ELSE
	Cmd_R:=3;
END_CASE
END_ACTION
ACTION Command:
(* Default response OK/NODATA *)
Cmd_R:=0;
Cmd_RLen:=0;
TxLen:=16;

(* Check object *)
CASE Cmd_Obj OF

	EO_SYS:
		Cmd_SYS();
(*
	EO_GRU:
		Cmd_GRU();

	EO_PDC:
		Cmd_PDC();
*)
	EO_CAL:
		Cmd_CAL();

	EO_CRON:
		Cmd_CRON();

	EO_VRD:
		Cmd_VRD();

ELSE
	Cmd_R:=1;
END_CASE

(* Generate response *)
IF TxLen>0 THEN
	RAWTOHEX(ADR(Cmd_Obj)	,2,ADR(TxData[ 0]));
	RAWTOHEX(ADR(Cmd_ObjIdx),2,ADR(TxData[ 4]));
	RAWTOHEX(ADR(Cmd_R)		,2,ADR(TxData[ 8]));
	RAWTOHEX(ADR(Cmd_RLen)	,2,ADR(TxData[12]));
	TxTrig:=TRUE;
END_IF
END_ACTION

(* POU Utils Functions/TCPSERVER, ST *)
FUNCTION_BLOCK TCPSERVER
(***********************************************************************************************************	*)
(* Version: 1.6                                    			          											*)
(* Date: 11.02.2011                                   					          							    *)
(***********************************************************************************************************	*)
(* WAGO Kontakttechnik GmbH Hansastr. 27 32423 Minden(Westf.)													*)
(* Tel. +0049 571/887-0 Fax. +0049 571/887-0																	*)
(* Author: VB																									*)
(***********************************************************************************************************	*)
(*Description:	A TCP server to read and write data													       		*)
(*Historie:																										*)
(*Version 1.6: 11.02.2011: Changes according to 750-880/881											 			*)
(*Version 1.5: 27.11.2008 Bugfix allow reuse port																*)
(*Version 1.4: 13.10.2008 Bugfix transmitting large data														*)
(*Version 1.3: 15.01.2007 Changes according to FW11																*)
(*Version 1.2: 09.03.2006 Changes for socket handle 0											       			*)
(*Version 1.1: 14.02.2005 Release																				*)
(***********************************************************************************************************	*)
VAR CONSTANT
	STATE_INIT     				 : BYTE:= 0;
	STATE_OPEN     				 : BYTE:= 1;
	STATE_TX       				 : BYTE:= 20;
	STATE_RX       				 : BYTE:= 30;
	STATE_CLOSE    				 : BYTE:= 40;
	STATE_ERROR_TRAP		 	 : BYTE:= 200;
END_VAR
VAR_INPUT
	xEnable    					: BOOL;	 (* Set TRUE to enable function block *)
	wPortNumber					: WORD;  (* Port *)
	tServerTimeOut				: TIME:=t#50s;
	ptSendData					: POINTER TO ARRAY[0..MAX_SEND_TCP_SERVER] OF BYTE;
	diSendCount					: DINT;
END_VAR
VAR_OUTPUT
	xClientConnected  			: BOOL:= FALSE;
	diError 					: DINT:= 0;
END_VAR
(* Status Codes -----------------------------------------
	16#8001 => No socket descriptor available 
	16#8002 => SysSockBind fails 
	16#8003 => SysSockListen fails 
	16#8004 => switching to none blocking mode fails
	16#8005 => SysSockClose() returns FALSE 
    16#8006 => SysSockConnect() fails
    16#8007 => SysSockSend() fails
	16#8008 => error state machine 
	16#8009 => timeout while waiting for data from server 
	16#0001 => server waiting for client to establish connection
------------------------------------------------------------*)
VAR_IN_OUT
	xStartSend					: BOOL;
	aReceiveBuffer				: ARRAY [0..MAX_RECEIVE_TCP_SERVER] OF BYTE;
	diReceiveCount				: DINT;
END_VAR

VAR
	m_State    					: BYTE:= 0;
	m_ReceiveBuffer				: ARRAY [0..MAX_RECEIVE_TCP_SERVER_SOCKET] OF BYTE;
	m_ServerSocket				: DINT:= SOCKET_INVALID;
	m_Socket					: DINT:= SOCKET_INVALID;
	m_AddressInfo				: SOCKADDRESS;
	m_BytesReceived				: DINT;
	m_diReturn					: DINT;
	m_xReturn					: BOOL;
	m_SizeSockadr				: DWORD;
	m_ConnectionWatchdog		: TON;
	m_Flags						: DINT;
	m_NoneBlocking   			: DINT:= 1;
	m_Blocking   				: DINT:= 0;
	i							: INT;
	m_count						: DINT;
	diOption					: DINT := 1;
	on: DINT;
END_VAR
IF xEnable THEN
	CASE m_State OF
		STATE_INIT:
			(* Create Socket *)
			m_ServerSocket:= SysSockCreate( SOCKET_AF_INET, SOCKET_STREAM, 0);
			IF m_ServerSocket = SOCKET_INVALID THEN
				(* *)
				diError:= 16#8001;
				m_State:= STATE_ERROR_TRAP;
				RETURN;
			ELSE
				;
			END_IF
			(* Address bindings *)
			(********************)
			on:=1;
			SysSockSetOption( m_ServerSocket, SOCKET_SOL, SOCKET_SO_REUSEADDR, ADR(on), SIZEOF(on) );

			m_AddressInfo.sin_family:= SOCKET_AF_INET;
			m_AddressInfo.sin_port  := SysSockHtons( wPortNumber);
			m_AddressInfo.sin_addr  := SOCKET_INADDR_ANY;
			IF NOT SysSockBind( m_ServerSocket, ADR(m_AddressInfo), SIZEOF(m_AddressInfo)) THEN
				diError:= 16#8002;
				m_State:= STATE_ERROR_TRAP;
				RETURN;
			END_IF
			(* Wait for connections *)
			(************************)
			IF NOT SysSockListen( m_ServerSocket, 1) THEN
				diError:= 16#8003;
				m_State:= STATE_ERROR_TRAP;
			END_IF

			(* Puts SOCKET in NonBlocking mode *)
			m_diReturn:= SysSockIoctl( m_ServerSocket, SOCKET_FIONBIO, ADR(m_NoneBlocking));

			m_State:= STATE_OPEN;


		STATE_OPEN: 	(* Waiting for incomming connection *)
				m_SizeSockadr:=SIZEOF(m_AddressInfo);
				m_Socket:= SysSockAccept( m_ServerSocket, ADR(m_AddressInfo), ADR(m_SizeSockadr));
				diError:=State_open;
				IF m_Socket <> SOCKET_INVALID THEN
					xClientConnected:=TRUE;
					(*Set Push-Bit:new V1.5*)
					IF ADR(%MW0)=16#30000000  OR ADR(%MW0)=16#20000000 THEN (*841 or 881*)
						SysSockSetOption(
							diSocket:=m_Socket,
							diLevel:=6,
							diOption:=SOCKET_TCP_NODELAY,
							pOptionValue:=ADR(diOption),
							diOptionLength:=SIZEOF(diOption));
					ELSE
							;
					END_IF
					SysSockIoctl( m_Socket, SOCKET_FIONBIO, ADR(m_NoneBlocking));
					m_State:= STATE_RX;
					diError:=0;
				END_IF

		STATE_RX:
					m_BytesReceived:= SysSockRecv( m_Socket, ADR(m_ReceiveBuffer), SIZEOF(m_ReceiveBuffer), 0);
					CASE m_BytesReceived OF
					-1:(*no data available or error occured*)
						m_ConnectionWatchdog(IN:=TRUE , PT:=tServerTimeOut );
						IF m_connectionWatchdog.Q THEN
							m_State:= STATE_CLOSE;
							m_ConnectionWatchdog(IN:=FALSE);(*reset connection watchdog*)
							diError := 16#8009;
						END_IF
					0:(* socket was "gracefully closed"  *)
						m_State:= STATE_CLOSE;
						diError := 16#8003;
					ELSE
						(* Copy received data into receive buffer *)
						(********************************)
						FOR i:= 0 TO DINT_TO_INT(m_BytesReceived	)-1 DO
							aReceiveBuffer[diReceiveCount]:= m_ReceiveBuffer[i];
							diReceiveCount:=(diReceiveCount+1) MOD SIZEOF(aReceiveBuffer);
						END_FOR

						m_ConnectionWatchdog(IN:=FALSE);(*reset connection watchdog*)
					END_CASE

				(*send data*)
				IF xStartSend	 THEN
					m_State := STATE_TX;
				END_IF

	STATE_TX:	 (* send TCP-message *)
		m_diReturn := SysSockSend(diSocket := m_Socket,
								  pbyBuffer := ADR(ptSendData^[m_count]),(*geändert V1.4 bisher: [0] *)
								  diBufferSize := diSendCount-m_count,
								  diFlags :=m_Flags);
		CASE m_diReturn OF
		-1:	(* ERROR or data could not yet be send (V1.3 due to new FW11) *)
			m_ConnectionWatchdog(IN:=TRUE , PT:=tServerTimeOut );
			IF m_connectionWatchdog.Q THEN
				m_State:= STATE_CLOSE;
				m_ConnectionWatchdog(IN:=FALSE);(*reset connection watchdog*)
				diError := 16#8007;
			END_IF
		0: (* socket was "gracefully closed"  *)
			m_State := STATE_CLOSE;
			diError := 16#8003;
		ELSE (* succesful *)
			m_count:=m_count+m_diReturn;
			IF m_count>=diSendCount THEN
				diError := 16#0000;
				m_State := STATE_RX;
				m_count:=0;
				xStartSend:=FALSE;
			END_IF
			m_ConnectionWatchdog(IN:=FALSE);(*reset connection watchdog*)
		END_CASE


		STATE_CLOSE:	(* Close the server *)

		IF ADR(%MW0)=16#30000000  OR ADR(%MW0)=16#20000000 THEN (*841 or 881*)
			;
		ELSE
			IF m_Socket>=0 THEN
				SysSockShutdown(m_Socket, 0);;(*870*)
			END_IF
		END_IF
		IF m_Socket>=0 THEN
			SysSockClose( m_Socket);
		END_IF
		xClientConnected:= FALSE;
		m_State:= STATE_OPEN; (* Try to open the server again *)
		m_ConnectionWatchdog(IN:=FALSE);(*reset connection watchdog*)

		STATE_ERROR_TRAP: (* Error Read/Write socket  *)
			m_State:= STATE_ERROR_TRAP;

	ELSE  (* Bad FSM code trap  *)
			m_State:= STATE_ERROR_TRAP;
			diError:= 16#8008;
	END_CASE;
ELSE
	IF m_State <> STATE_INIT THEN
		IF ADR(%MW0)=16#30000000  OR ADR(%MW0)=16#20000000 THEN (*841 or 881*)
			;
		ELSE
			IF m_Socket>=0 THEN
				SysSockShutdown(m_Socket, 0);;(*870*)
			END_IF
		END_IF
		IF m_Socket>=0 THEN
			SysSockClose( m_Socket);
		END_IF
		IF ADR(%MW0)=16#30000000  OR ADR(%MW0)=16#20000000 THEN (*841 or 881*)
			;
		ELSE
			IF m_ServerSocket>=0 THEN
				SysSockShutdown(m_ServerSocket, 0);;(*870*)
			END_IF
		END_IF
		IF m_ServerSocket>=0 THEN
			SysSockClose( m_ServerSocket);
		END_IF
		xClientConnected:= FALSE;
		diError:= 0;
		m_State:= STATE_init; (* Try to open the server again *)
		m_ConnectionWatchdog(IN:=FALSE);(*reset connection watchdog*)
	END_IF
END_IF
END_FUNCTION_BLOCK

(* POU Utils Functions/HEXTORAW, ST *)
FUNCTION HEXTORAW : WORD
VAR_INPUT
	pString		: POINTER TO BYTE;
	StringLen	: WORD;
	pData		: POINTER TO BYTE;
END_VAR
VAR
	xl: WORD;
	xi: WORD;
	xr: BYTE;
END_VAR
xl:=0;
xi:=0;

WHILE xi<StringLen DO

	IF pString^>=97 AND pString^<=102 THEN
		xr := pString^ - 87;
	ELSIF pString^>=65 AND pString^<=70 THEN
		xr := pString^ - 55;
	ELSIF pString^>=48 AND pString^<=57 THEN
		xr := pString^ - 48;
	ELSE
		xr := 16;
	END_IF

	IF xr<16 THEN
		IF (xi AND 1)=0 THEN
			pData^ := xr * 16;
		ELSE
			pData^ := pData^ + xr;
			pData := pData + 1;
			xl := xl + 1;
		END_IF
	END_IF

	xi := xi + 1;
	pString := pString + 1;

END_WHILE

HEXTORAW:=xl;
END_FUNCTION

(* POU Utils Functions/RAWTOHEX, ST *)
FUNCTION RAWTOHEX : WORD
VAR_INPUT
	pData: POINTER TO BYTE;
	DataLen: WORD;
	pString: POINTER TO BYTE;
END_VAR
VAR
	xl: WORD;
END_VAR
xl:=0;

WHILE DataLen>0 DO

	pString^ := (pData^ / 16#10) + 48 + (((pData^ / 16#10)/10)*7);
	pString:=pString+1;
	pString^ := (pData^ AND 16#0F)  + 48 + (((pData^ AND 16#0F)/10)*7);
	pString:=pString+1;
	pData:=pData+1;
	DataLen:=DataLen-1;
	xl:=xl+2;

END_WHILE

(*pString^:=0;*)

RAWTOHEX:=xl;
END_FUNCTION

(* POU Utils/USRLED_Update, ST *)
PROGRAM USRLED_Update
VAR
	OldStatus: en_SYS_Status;

	aFS : ARRAY [0..24] OF FLASHING_SEQUENCE :=
		(Colour:=GREEN,  Frequency:=1,   Relation:=128, Duration:=t#0s,    NextIndex:=0),  (* 0 => RUNNING *)
		(Colour:=ORANGE, Frequency:=1,   Relation:=128, Duration:=t#0s,    NextIndex:=1),  (* 1 => INIT *)
		(Colour:=RED,    Frequency:=4,   Relation:=128, Duration:=t#0s,    NextIndex:=2),  (* 2 => ERROR *)
		(Colour:=RED,    Frequency:=10,  Relation:=128, Duration:=t#0s,    NextIndex:=3),  (* 3 => ALARM *)
		(Colour:=ORANGE, Frequency:=200, Relation:=16,  Duration:=t#100ms, NextIndex:=11), (* 10 *)
		(Colour:=ORANGE, Frequency:=200, Relation:=32,  Duration:=t#100ms, NextIndex:=12),
		(Colour:=ORANGE, Frequency:=200, Relation:=64,  Duration:=t#100ms, NextIndex:=13),
		(Colour:=ORANGE, Frequency:=200, Relation:=128, Duration:=t#100ms, NextIndex:=14),
		(Colour:=ORANGE, Frequency:=200, Relation:=192, Duration:=t#100ms, NextIndex:=15),
		(Colour:=ORANGE, Frequency:=200, Relation:=128, Duration:=t#100ms, NextIndex:=16),
		(Colour:=ORANGE, Frequency:=200, Relation:=64,  Duration:=t#100ms, NextIndex:=17),
		(Colour:=ORANGE, Frequency:=200, Relation:=32,  Duration:=t#100ms, NextIndex:=18),
		(Colour:=ORANGE, Frequency:=200, Relation:=16,  Duration:=t#100ms, NextIndex:=19),
		(Colour:=ORANGE, Frequency:=200, Relation:=8,   Duration:=t#100ms, NextIndex:=10),
		(Colour:=GREEN,  Frequency:=200, Relation:=16,  Duration:=t#100ms, NextIndex:=21), (* 20 *)
		(Colour:=GREEN,  Frequency:=200, Relation:=32,  Duration:=t#100ms, NextIndex:=22),
		(Colour:=GREEN,  Frequency:=200, Relation:=64,  Duration:=t#100ms, NextIndex:=23),
		(Colour:=GREEN,  Frequency:=200, Relation:=128, Duration:=t#100ms, NextIndex:=24),
		(Colour:=GREEN,  Frequency:=200, Relation:=192, Duration:=t#100ms, NextIndex:=25),
		(Colour:=GREEN,  Frequency:=200, Relation:=128, Duration:=t#100ms, NextIndex:=26),
		(Colour:=GREEN,  Frequency:=200, Relation:=64,  Duration:=t#100ms, NextIndex:=27),
		(Colour:=GREEN,  Frequency:=200, Relation:=32,  Duration:=t#100ms, NextIndex:=28),
		(Colour:=GREEN,  Frequency:=200, Relation:=16,  Duration:=t#100ms, NextIndex:=29),
		(Colour:=GREEN,  Frequency:=200, Relation:=8,   Duration:=t#100ms, NextIndex:=20);

	pFS : POINTER TO FLASHING_SEQUENCE;


END_VAR
IF Sys.Status <> OldStatus THEN

	OldStatus:=Sys.Status;

	CASE OldStatus OF

		S_STARTUP:
			pFS:=ADR(aFS);
			SET_FLASHING_SEQUENCE(EN:=TRUE, POINTER_TO_POINTER_TO_ARRAY:=ADR(pFS));
			SET_FLASHING_SEQUENCE_INDEX(EN:=TRUE, IMMEDIATE:=FALSE, INDEX:=1);
			START_FLASHING_SEQUENCE(EN:=TRUE);

		S_RUNNING:
			SET_FLASHING_SEQUENCE_INDEX(EN:=TRUE, IMMEDIATE:=TRUE, INDEX:=0);

	END_CASE

END_IF
END_PROGRAM

(* POU Utils/CSV_Log, ST *)
FUNCTION CSV_Log : BOOL
VAR_INPUT
END_VAR
VAR CONSTANT
	LogFileName:STRING:='S:\LOGS_ID4V3.CSV';
END_VAR
VAR
	s1 : STRING(256);
	hFile: 	DWORD;
END_VAR
(* Check file presence *)
hFile:=SysFileOpen(LogFileName,'r');
IF hFile=0 THEN
	(*** File not exist *** Create file and write header *)
	hFile:=SysFileOpen(LogFileName,'w');
	IF hFile<>0 THEN
		(* Write CSV header *)
		s1:='Title1;Title2,...';
		SysFileWrite(hFile, ADR(s1), LEN(s1));
		SysFileWrite(hFile, ADR(Logger_CRLF), LEN(Logger_CRLF));
	END_IF
ELSE
	(*** File exist *** Close file and reopen in append mode *)
	SysFileClose(hFile);
	hFile:=SysFileOpen(LogFileName,'a');
END_IF

(* Log to file *)
IF hFile<>0 THEN
	(* Date stamp *)
	s1:=REPLACE( Sys.Time_LogString , ' ' , 1 , 11 );
	SysFileWrite(hFile, ADR(s1), LEN(s1));
	(* Write CSV data *)
	s1:=CONCAT(';', 'Data1' );
	s1:=CONCAT(s1 , ';');
	s1:=CONCAT(s1 , 'Data2' );
	s1:=CONCAT(s1 , ';');
	s1:=CONCAT(s1 , '...' );
	SysFileWrite(hFile, ADR(s1), LEN(s1));
	(* Add line CRLF and close *)
	SysFileWrite(hFile, ADR(Logger_CRLF), LEN(Logger_CRLF));
	SysFileClose(hFile);
END_IF
END_FUNCTION

(* POU CLV/CLV__Cmd, ST *)
PROGRAM CLV__Cmd
(* === Execute server command ===
   v1.0[27/05/15]
*)
VAR_INPUT
END_VAR
VAR_OUTPUT
	Cmd_R
	Cmd_RLen
END_VAR
VAR
END_VAR
(* Default response OK/NODATA *)
Cmd_R:=0;
Cmd_RLen:=0;
TxLen:=16;

(* Check object *)
CASE Cmd_Obj OF

	EO_SYS:
		Cmd_SYS();
(*
	EO_GRU:
		Cmd_GRU();

	EO_PDC:
		Cmd_PDC();

	EO_CAL:
		Cmd_CAL();

	EO_CRON:
		Cmd_CRON();
*)
ELSE
	Cmd_R:=1;
END_CASE
END_PROGRAM

(* POU CLV/CLV__LogTrig, ST *)
PROGRAM CLV__LogTrig
(* === Log regular informations ===
   v1.0[27/05/15]
*)
VAR
	s1 : STRING(160);
	i  : BYTE;
END_VAR
(*---------------------------------------------------------------*)
	CLV.LogHead();
(*---------------------------------------------------------------*)

(*** PROJECT SPECIFIC CODE HERE ***)

(*---------------------------------------------------------------*)
	CLV.LogSend();
(*---------------------------------------------------------------*)
END_PROGRAM

(* POU Plant/SCA_Proc, ST *)
PROGRAM SCA_Proc
VAR
	SCA01_5			:FLT_TAP;
	SCA01_6			:FLT_TAP;

	SCA02_1			:FLT_TAP;
	SCA02_2			:FLT_TAP;
	SCA02_3			:FLT_TAP;
	SCA02_4			:FLT_TAP;
	SCA02_5			:FLT_TAP;
	SCA02_6			:FLT_TAP;
	SCA02_7			:FLT_TAP;
	SCA02_8			:FLT_TAP;
	SCA02_9			:FLT_TAP;

	SCA03_1			:FLT_TAP;
	SCA03_2			:FLT_TAP;
	SCA03_3			:FLT_TAP;
	SCA03_4			:FLT_TAP;
	SCA03_5			:FLT_TAP;
	SCA03_6			:FLT_TAP;
	SCA03_7			:FLT_TAP;
	SCA03_8			:FLT_TAP;
	SCA03_9			:FLT_TAP;
	SCA03_10		:FLT_TAP;
	SCA03_11		:FLT_TAP;
	SCA03_12		:FLT_TAP;
	SCA03_13		:FLT_TAP;
	SCA03_14		:FLT_TAP;
	SCA03_15		:FLT_TAP;
	SCA03_16		:FLT_TAP;
	SCA03_17		:FLT_TAP;
	SCA03_18		:FLT_TAP;
	SCA03_19		:FLT_TAP;
	SCA03_20		:FLT_TAP;
	SCA03_21		:FLT_TAP;
	SCA03_22		:FLT_TAP;

END_VAR
(***** SCA01 *****)
SCA01_1_DO:=SCA01_6.OUT;

SCA01_2_DO:=SCA02_1.OUT;

SCA01_3_DO:=SCA02_2.OUT  OR SCA02_3.OUT  OR SCA02_4.OUT  OR SCA02_5.OUT  OR SCA02_6.OUT  OR
			SCA02_7.OUT  OR SCA02_8.OUT  OR SCA02_9.OUT;

SCA01_4_DO:=SCA03_1.OUT  OR SCA03_2.OUT  OR SCA03_3.OUT  OR SCA03_4.OUT  OR SCA03_5.OUT  OR
			SCA03_6.OUT  OR SCA03_7.OUT  OR SCA03_8.OUT  OR SCA03_9.OUT  OR SCA03_10.OUT OR
			SCA03_11.OUT OR SCA03_12.OUT OR SCA03_13.OUT OR SCA03_14.OUT OR SCA03_15.OUT OR
			SCA03_16.OUT OR SCA03_17.OUT OR SCA03_18.OUT OR SCA03_19.OUT OR SCA03_20.OUT OR
			SCA03_21.OUT OR SCA03_22.OUT;

SCA01_5(IN:=SCA01_5_DI);
IF SCA01_5.EVL THEN LogEv(EL_Wrn,EO_SCA,1,1,'5'); END_IF
IF SCA01_5.EVH THEN	LogEv(EL_Log,EO_SCA,1,2,'5'); END_IF

SCA01_6(IN:=SCA01_6_DI);
IF SCA01_6.EVL THEN	LogEv(EL_Wrn,EO_SCA,1,1,'6'); END_IF
IF SCA01_6.EVH THEN	LogEv(EL_Log,EO_SCA,1,2,'6'); END_IF

(***** SCA02 *****)

SCA02_1(IN:=SCA02_1_DI);
IF SCA02_1.EVL THEN	LogEv(EL_Wrn,EO_SCA,2,1,'1'); END_IF
IF SCA02_1.EVH THEN	LogEv(EL_Log,EO_SCA,2,2,'1'); END_IF
SCA02_2(IN:=SCA02_2_DI);
IF SCA02_2.EVL THEN	LogEv(EL_Wrn,EO_SCA,2,1,'2'); END_IF
IF SCA02_2.EVH THEN	LogEv(EL_Log,EO_SCA,2,2,'2'); END_IF
SCA02_3(IN:=SCA02_3_DI);
IF SCA02_3.EVL THEN	LogEv(EL_Wrn,EO_SCA,2,1,'3'); END_IF
IF SCA02_3.EVH THEN	LogEv(EL_Log,EO_SCA,2,2,'3'); END_IF
SCA02_4(IN:=SCA02_4_DI);
IF SCA02_4.EVL THEN	LogEv(EL_Wrn,EO_SCA,2,1,'4'); END_IF
IF SCA02_4.EVH THEN	LogEv(EL_Log,EO_SCA,2,2,'4'); END_IF
SCA02_5(IN:=SCA02_5_DI);
IF SCA02_5.EVL THEN	LogEv(EL_Wrn,EO_SCA,2,1,'5'); END_IF
IF SCA02_5.EVH THEN	LogEv(EL_Log,EO_SCA,2,2,'5'); END_IF
SCA02_6(IN:=SCA02_6_DI);
IF SCA02_6.EVL THEN	LogEv(EL_Wrn,EO_SCA,2,1,'6'); END_IF
IF SCA02_6.EVH THEN	LogEv(EL_Log,EO_SCA,2,2,'6'); END_IF
SCA02_7(IN:=SCA02_7_DI);
IF SCA02_7.EVL THEN	LogEv(EL_Wrn,EO_SCA,2,1,'7'); END_IF
IF SCA02_7.EVH THEN	LogEv(EL_Log,EO_SCA,2,2,'7'); END_IF
SCA02_8(IN:=SCA02_8_DI);
IF SCA02_8.EVL THEN	LogEv(EL_Wrn,EO_SCA,2,1,'8'); END_IF
IF SCA02_8.EVH THEN	LogEv(EL_Log,EO_SCA,2,2,'8'); END_IF
SCA02_9(IN:=SCA02_9_DI);
IF SCA02_9.EVL THEN	LogEv(EL_Wrn,EO_SCA,2,1,'9'); END_IF
IF SCA02_9.EVH THEN	LogEv(EL_Log,EO_SCA,2,2,'9'); END_IF

(***** SCA03 *****)

SCA03_1(IN:=SCA03_1_DI);
IF SCA03_1.EVL THEN	LogEv(EL_Wrn,EO_SCA,3,1,'1'); END_IF
IF SCA03_1.EVH THEN	LogEv(EL_Log,EO_SCA,3,2,'1'); END_IF
SCA03_2(IN:=SCA03_2_DI);
IF SCA03_2.EVL THEN	LogEv(EL_Wrn,EO_SCA,3,1,'2'); END_IF
IF SCA03_2.EVH THEN	LogEv(EL_Log,EO_SCA,3,2,'2'); END_IF
SCA03_3(IN:=SCA03_3_DI);
IF SCA03_3.EVL THEN	LogEv(EL_Wrn,EO_SCA,3,1,'3'); END_IF
IF SCA03_3.EVH THEN	LogEv(EL_Log,EO_SCA,3,2,'3'); END_IF
SCA03_4(IN:=SCA03_4_DI);
IF SCA03_4.EVL THEN	LogEv(EL_Wrn,EO_SCA,3,1,'4'); END_IF
IF SCA03_4.EVH THEN	LogEv(EL_Log,EO_SCA,3,2,'4'); END_IF
SCA03_5(IN:=SCA03_5_DI);
IF SCA03_5.EVL THEN	LogEv(EL_Wrn,EO_SCA,3,1,'5'); END_IF
IF SCA03_5.EVH THEN	LogEv(EL_Log,EO_SCA,3,2,'5'); END_IF
SCA03_6(IN:=SCA03_6_DI);
IF SCA03_6.EVL THEN	LogEv(EL_Wrn,EO_SCA,3,1,'6'); END_IF
IF SCA03_6.EVH THEN	LogEv(EL_Log,EO_SCA,3,2,'6'); END_IF
SCA03_7(IN:=SCA03_7_DI);
IF SCA03_7.EVL THEN	LogEv(EL_Wrn,EO_SCA,3,1,'7'); END_IF
IF SCA03_7.EVH THEN	LogEv(EL_Log,EO_SCA,3,2,'7'); END_IF
SCA03_8(IN:=SCA03_8_DI);
IF SCA03_8.EVL THEN	LogEv(EL_Wrn,EO_SCA,3,1,'8'); END_IF
IF SCA03_8.EVH THEN	LogEv(EL_Log,EO_SCA,3,2,'8'); END_IF
SCA03_9(IN:=SCA03_9_DI);
IF SCA03_9.EVL THEN	LogEv(EL_Wrn,EO_SCA,3,1,'9'); END_IF
IF SCA03_9.EVH THEN	LogEv(EL_Log,EO_SCA,3,2,'9'); END_IF
SCA03_10(IN:=SCA03_10_DI);
IF SCA03_10.EVL THEN	LogEv(EL_Wrn,EO_SCA,3,1,'10'); END_IF
IF SCA03_10.EVH THEN	LogEv(EL_Log,EO_SCA,3,2,'10'); END_IF
SCA03_11(IN:=SCA03_11_DI);
IF SCA03_11.EVL THEN	LogEv(EL_Wrn,EO_SCA,3,1,'11'); END_IF
IF SCA03_11.EVH THEN	LogEv(EL_Log,EO_SCA,3,2,'11'); END_IF
SCA03_12(IN:=SCA03_12_DI);
IF SCA03_12.EVL THEN	LogEv(EL_Wrn,EO_SCA,3,1,'12'); END_IF
IF SCA03_12.EVH THEN	LogEv(EL_Log,EO_SCA,3,2,'12'); END_IF
SCA03_13(IN:=SCA03_13_DI);
IF SCA03_13.EVL THEN	LogEv(EL_Wrn,EO_SCA,3,1,'13'); END_IF
IF SCA03_13.EVH THEN	LogEv(EL_Log,EO_SCA,3,2,'13'); END_IF
SCA03_14(IN:=SCA03_14_DI);
IF SCA03_14.EVL THEN	LogEv(EL_Wrn,EO_SCA,3,1,'14'); END_IF
IF SCA03_14.EVH THEN	LogEv(EL_Log,EO_SCA,3,2,'14'); END_IF
SCA03_15(IN:=SCA03_15_DI);
IF SCA03_15.EVL THEN	LogEv(EL_Wrn,EO_SCA,3,1,'15'); END_IF
IF SCA03_15.EVH THEN	LogEv(EL_Log,EO_SCA,3,2,'15'); END_IF
SCA03_16(IN:=SCA03_16_DI);
IF SCA03_16.EVL THEN	LogEv(EL_Wrn,EO_SCA,3,1,'16'); END_IF
IF SCA03_16.EVH THEN	LogEv(EL_Log,EO_SCA,3,2,'16'); END_IF
SCA03_17(IN:=SCA03_17_DI);
IF SCA03_17.EVL THEN	LogEv(EL_Wrn,EO_SCA,3,1,'17'); END_IF
IF SCA03_17.EVH THEN	LogEv(EL_Log,EO_SCA,3,2,'17'); END_IF
SCA03_18(IN:=SCA03_18_DI);
IF SCA03_18.EVL THEN	LogEv(EL_Wrn,EO_SCA,3,1,'18'); END_IF
IF SCA03_18.EVH THEN	LogEv(EL_Log,EO_SCA,3,2,'18'); END_IF
SCA03_19(IN:=SCA03_19_DI);
IF SCA03_19.EVL THEN	LogEv(EL_Wrn,EO_SCA,3,1,'19'); END_IF
IF SCA03_19.EVH THEN	LogEv(EL_Log,EO_SCA,3,2,'19'); END_IF
SCA03_20(IN:=SCA03_20_DI);
IF SCA03_20.EVL THEN	LogEv(EL_Wrn,EO_SCA,3,1,'20'); END_IF
IF SCA03_20.EVH THEN	LogEv(EL_Log,EO_SCA,3,2,'20'); END_IF
SCA03_21(IN:=SCA03_21_DI);
IF SCA03_21.EVL THEN	LogEv(EL_Wrn,EO_SCA,3,1,'21'); END_IF
IF SCA03_21.EVH THEN	LogEv(EL_Log,EO_SCA,3,2,'21'); END_IF
SCA03_22(IN:=SCA03_22_DI);
IF SCA03_22.EVL THEN	LogEv(EL_Wrn,EO_SCA,3,1,'22'); END_IF
IF SCA03_22.EVH THEN	LogEv(EL_Log,EO_SCA,3,2,'22'); END_IF
END_PROGRAM
ACTION AddLogData:
Logger.s1:='&SCA01=';
Logger.s1:=CONCAT(Logger.s1,BYTE_TO_STRING(BOOL_TO_BYTE(SCA01_1_DO))		); Logger.s1:=CONCAT(Logger.s1,';');
Logger.s1:=CONCAT(Logger.s1,BYTE_TO_STRING(BOOL_TO_BYTE(SCA01_2_DO))		); Logger.s1:=CONCAT(Logger.s1,';');
Logger.s1:=CONCAT(Logger.s1,BYTE_TO_STRING(BOOL_TO_BYTE(SCA01_3_DO))		); Logger.s1:=CONCAT(Logger.s1,';');
Logger.s1:=CONCAT(Logger.s1,BYTE_TO_STRING(BOOL_TO_BYTE(SCA01_4_DO))		); Logger.s1:=CONCAT(Logger.s1,';');
Logger.s1:=CONCAT(Logger.s1,BYTE_TO_STRING(BOOL_TO_BYTE(SCA01_5.OUT))		); Logger.s1:=CONCAT(Logger.s1,';');
Logger.s1:=CONCAT(Logger.s1,BYTE_TO_STRING(BOOL_TO_BYTE(SCA01_6.OUT))		);
ADDSTRING(ADR(Logger.TData), ADR(Logger.s1), Logger.TLen);

Logger.s1:='&SCA02=';
Logger.s1:=CONCAT(Logger.s1,BYTE_TO_STRING(BOOL_TO_BYTE(SCA02_1.OUT))		); Logger.s1:=CONCAT(Logger.s1,';');
Logger.s1:=CONCAT(Logger.s1,BYTE_TO_STRING(BOOL_TO_BYTE(SCA02_2.OUT))		); Logger.s1:=CONCAT(Logger.s1,';');
Logger.s1:=CONCAT(Logger.s1,BYTE_TO_STRING(BOOL_TO_BYTE(SCA02_3.OUT))		); Logger.s1:=CONCAT(Logger.s1,';');
Logger.s1:=CONCAT(Logger.s1,BYTE_TO_STRING(BOOL_TO_BYTE(SCA02_4.OUT))		); Logger.s1:=CONCAT(Logger.s1,';');
Logger.s1:=CONCAT(Logger.s1,BYTE_TO_STRING(BOOL_TO_BYTE(SCA02_5.OUT))		); Logger.s1:=CONCAT(Logger.s1,';');
Logger.s1:=CONCAT(Logger.s1,BYTE_TO_STRING(BOOL_TO_BYTE(SCA02_6.OUT))		); Logger.s1:=CONCAT(Logger.s1,';');
Logger.s1:=CONCAT(Logger.s1,BYTE_TO_STRING(BOOL_TO_BYTE(SCA02_7.OUT))		); Logger.s1:=CONCAT(Logger.s1,';');
Logger.s1:=CONCAT(Logger.s1,BYTE_TO_STRING(BOOL_TO_BYTE(SCA02_8.OUT))		); Logger.s1:=CONCAT(Logger.s1,';');
Logger.s1:=CONCAT(Logger.s1,BYTE_TO_STRING(BOOL_TO_BYTE(SCA02_9.OUT))		);
ADDSTRING(ADR(Logger.TData), ADR(Logger.s1), Logger.TLen);

Logger.s1:='&SCA03=';
Logger.s1:=CONCAT(Logger.s1,BYTE_TO_STRING(BOOL_TO_BYTE(SCA03_1.OUT))		); Logger.s1:=CONCAT(Logger.s1,';');
Logger.s1:=CONCAT(Logger.s1,BYTE_TO_STRING(BOOL_TO_BYTE(SCA03_2.OUT))		); Logger.s1:=CONCAT(Logger.s1,';');
Logger.s1:=CONCAT(Logger.s1,BYTE_TO_STRING(BOOL_TO_BYTE(SCA03_3.OUT))		); Logger.s1:=CONCAT(Logger.s1,';');
Logger.s1:=CONCAT(Logger.s1,BYTE_TO_STRING(BOOL_TO_BYTE(SCA03_4.OUT))		); Logger.s1:=CONCAT(Logger.s1,';');
Logger.s1:=CONCAT(Logger.s1,BYTE_TO_STRING(BOOL_TO_BYTE(SCA03_5.OUT))		); Logger.s1:=CONCAT(Logger.s1,';');
Logger.s1:=CONCAT(Logger.s1,BYTE_TO_STRING(BOOL_TO_BYTE(SCA03_6.OUT))		); Logger.s1:=CONCAT(Logger.s1,';');
Logger.s1:=CONCAT(Logger.s1,BYTE_TO_STRING(BOOL_TO_BYTE(SCA03_7.OUT))		); Logger.s1:=CONCAT(Logger.s1,';');
Logger.s1:=CONCAT(Logger.s1,BYTE_TO_STRING(BOOL_TO_BYTE(SCA03_8.OUT))		); Logger.s1:=CONCAT(Logger.s1,';');
Logger.s1:=CONCAT(Logger.s1,BYTE_TO_STRING(BOOL_TO_BYTE(SCA03_9.OUT))		); Logger.s1:=CONCAT(Logger.s1,';');
Logger.s1:=CONCAT(Logger.s1,BYTE_TO_STRING(BOOL_TO_BYTE(SCA03_10.OUT))		); Logger.s1:=CONCAT(Logger.s1,';');
Logger.s1:=CONCAT(Logger.s1,BYTE_TO_STRING(BOOL_TO_BYTE(SCA03_11.OUT))		); Logger.s1:=CONCAT(Logger.s1,';');
Logger.s1:=CONCAT(Logger.s1,BYTE_TO_STRING(BOOL_TO_BYTE(SCA03_12.OUT))		); Logger.s1:=CONCAT(Logger.s1,';');
Logger.s1:=CONCAT(Logger.s1,BYTE_TO_STRING(BOOL_TO_BYTE(SCA03_13.OUT))		); Logger.s1:=CONCAT(Logger.s1,';');
Logger.s1:=CONCAT(Logger.s1,BYTE_TO_STRING(BOOL_TO_BYTE(SCA03_14.OUT))		); Logger.s1:=CONCAT(Logger.s1,';');
Logger.s1:=CONCAT(Logger.s1,BYTE_TO_STRING(BOOL_TO_BYTE(SCA03_15.OUT))		); Logger.s1:=CONCAT(Logger.s1,';');
Logger.s1:=CONCAT(Logger.s1,BYTE_TO_STRING(BOOL_TO_BYTE(SCA03_16.OUT))		); Logger.s1:=CONCAT(Logger.s1,';');
Logger.s1:=CONCAT(Logger.s1,BYTE_TO_STRING(BOOL_TO_BYTE(SCA03_17.OUT))		); Logger.s1:=CONCAT(Logger.s1,';');
Logger.s1:=CONCAT(Logger.s1,BYTE_TO_STRING(BOOL_TO_BYTE(SCA03_18.OUT))		); Logger.s1:=CONCAT(Logger.s1,';');
Logger.s1:=CONCAT(Logger.s1,BYTE_TO_STRING(BOOL_TO_BYTE(SCA03_19.OUT))		); Logger.s1:=CONCAT(Logger.s1,';');
Logger.s1:=CONCAT(Logger.s1,BYTE_TO_STRING(BOOL_TO_BYTE(SCA03_20.OUT))		); Logger.s1:=CONCAT(Logger.s1,';');
Logger.s1:=CONCAT(Logger.s1,BYTE_TO_STRING(BOOL_TO_BYTE(SCA03_21.OUT))		); Logger.s1:=CONCAT(Logger.s1,';');
Logger.s1:=CONCAT(Logger.s1,BYTE_TO_STRING(BOOL_TO_BYTE(SCA03_22.OUT))		);
ADDSTRING(ADR(Logger.TData), ADR(Logger.s1), Logger.TLen);
END_ACTION

(* POU Utils Functions/FLT_TAP, ST *)
FUNCTION_BLOCK FLT_TAP
VAR_INPUT
	IN		: BOOL;
	TAP		: BYTE:=4;
	INITEV	: BOOL:=TRUE;
END_VAR
VAR_OUTPUT
	OUT		: BOOL;
	EVH		: BOOL;
	EVL		: BOOL;
END_VAR
VAR
	init	: BOOL:=FALSE;
	cnt		: BYTE;
END_VAR
EVH:=FALSE;
EVL:=FALSE;

IF NOT init THEN
	init := TRUE;
	IF INITEV THEN
		OUT  := NOT IN;
		cnt  := TAP;
	ELSE
		OUT  := IN;
	END_IF
END_IF

IF OUT<>IN THEN
	cnt:=cnt+1;
	IF cnt>TAP THEN
		OUT:=IN;
		cnt:=0;
		IF OUT THEN EVH:=TRUE; ELSE EVL:=TRUE; END_IF
	END_IF
ELSE
	cnt:=0;
END_IF
END_FUNCTION_BLOCK

(* POU TCP_Logger/LogEv, ST *)
FUNCTION LogEv : BOOL
VAR_INPUT
	Level	: en_Logger_ErrLev;
	Object  : en_SYS_Objects;
	Index	: WORD;
	Error	: WORD;
	Message : STRING;
END_VAR
VAR
	s1 : STRING(160);
	i  : INT;
END_VAR
(* Execute error level operations *)
CASE Level OF
	EL_Wrn: 		Sys.Warning:=TRUE;
	EL_Alarm: 		Sys.Alarm  :=TRUE;
	EL_AlarmStop: 	Sys.Alarm  :=TRUE; (* GO TO STOP STATE!! *)
END_CASE

(* Fill lastlog list *)
s1:=CONCAT(Sys.Time_LogString,';Lev=');
s1:=CONCAT(s1,INT_TO_STRING(Level));
s1:=CONCAT(s1,';Obj=');
s1:=CONCAT(s1,INT_TO_STRING(Object));
s1:=CONCAT(s1,';Idx=');
s1:=CONCAT(s1,WORD_TO_STRING(Index));
s1:=CONCAT(s1,';Err=');
s1:=CONCAT(s1,WORD_TO_STRING(Error));
Sys.LastLogs_Dat[Sys.LastLogs_Idx]:=s1;
Sys.LastLogs_Msg[Sys.LastLogs_Idx]:=Message;
Sys.LastLogs_Idx:=Sys.LastLogs_Idx+1;
IF Sys.LastLogs_Idx>5 THEN Sys.LastLogs_Idx:=0; END_IF

(*---------------------------------------------------------------*)
	Logger_Head();
(*---------------------------------------------------------------*)

(* Insert ERR *)
s1:=CONCAT('&ERR=',INT_TO_STRING(Level));
s1:=CONCAT(s1,';');
s1:=CONCAT(s1,INT_TO_STRING(Object));
s1:=CONCAT(s1,';');
s1:=CONCAT(s1,WORD_TO_STRING(Index));
s1:=CONCAT(s1,';');
s1:=CONCAT(s1,WORD_TO_STRING(Error));
s1:=CONCAT(s1,';');
ADDSTRING(ADR(Logger.TData), ADR(s1), Logger.TLen);
s1:=Message;
STR_NOSPACES(ADR(s1));
ADDSTRING(ADR(Logger.TData), ADR(s1), Logger.TLen);

(*---------------------------------------------------------------*)
	Logger_Send();
(*---------------------------------------------------------------*)
END_FUNCTION

(* POU TCP_Logger/Logger_Head, ST *)
FUNCTION Logger_Head : BOOL
VAR
	s1 : STRING(160);
	i  : BYTE;
END_VAR
Logger.TLen:=0;
(* Set GET header *)
ADDSTRING(ADR(Logger.TData), ADR(Logger_GETSTART), Logger.TLen);

(* Insert Header *)
s1:=INSERT('ID=&V=1&D=',DWORD_TO_STRING(Plant_SN),3);
s1:=CONCAT(s1,Sys.Time_LogString);
s1:=CONCAT(s1,'&S=');
IF Sys.Alarm THEN i:=2; ELSIF Sys.Warning THEN i:=1; ELSE i:=0; END_IF
s1:=CONCAT(s1,BYTE_TO_STRING(i));
ADDSTRING(ADR(Logger.TData), ADR(s1), Logger.TLen);
END_FUNCTION

(* POU Utils Functions/ADDSTRING, ST *)
FUNCTION ADDSTRING : BOOL (* Append string to a byte buffer *)
VAR_INPUT
	pTxData: POINTER TO BYTE;
	pString: POINTER TO BYTE;
END_VAR
VAR_IN_OUT
	TxLen: DINT;
END_VAR
VAR
END_VAR
pTxData:=pTxData+TxLen;
WHILE pString^<>0 DO
	pTxData^:=pString^;
	pString:=pString+1;
	pTxData:=pTxData+1;
	TxLen:=TxLen+1;
END_WHILE
END_FUNCTION

(* POU Utils Functions/STR_NOSPACES, ST *)
FUNCTION STR_NOSPACES : BOOL (* Replace spaces and bad chars with allowed ones, used as HTTP-GET validator *)
VAR_INPUT
	pString: POINTER TO BYTE;
END_VAR
VAR
END_VAR
WHILE pString^<>0 DO
	IF pString^=16#20 (* space *) THEN pString^:=16#5F; (*'_'*) END_IF
	pString:=pString+1;
END_WHILE
END_FUNCTION

(* POU TCP_Logger/Logger_Send, ST *)
FUNCTION Logger_Send : BOOL
VAR
	hFile: 	DWORD;
	pos:	DWORD;
END_VAR
(* Finalize string *)
ADDSTRING(ADR(Logger.TData), ADR(Logger_GETEND), Logger.TLen);

(* Read log position *)
pos:=SysFileGetSize(Logger_DataFile);
(* Check log size, bckup and erase if no pending messages *)
IF pos>5000000(*5M*) THEN
	hFile:=SysFileOpen(Logger_IndexFile,'r');
	IF hFile=0 THEN
		SysFileDelete(Logger_DataFileOld);
		SysFileRename(Logger_DataFile,Logger_DataFileOld);
		pos:=0;
	ELSE
		SysFileClose(hFile);
	END_IF
END_IF
(* Write message on log file *)
hFile:=SysFileOpen(Logger_DataFile,'a');
IF hFile<>0 THEN
	SysFileWrite(hFile, ADR(Logger.TData), Logger.TLen);
	SysFileClose(hFile);
ELSE
	Sys.Warning:=TRUE;
END_IF


(* Check logger status *)
IF Logger.SendReq=FALSE THEN
	(* Set log position for recovery *)
	Logger.SendIdx:=pos;
	(* Copy message data *)
	MEMCPY(ADR(Logger.TData),ADR(Logger.SendData),DINT_TO_WORD(Logger.TLen));
	Logger.SendLen:=Logger.TLen;
	(* Trigger request *)
	Logger.SendReq:=TRUE;
ELSE
	(* Add message position+size in recovery indexes *)
	hFile:=SysFileOpen(Logger_IndexFile,'a');
	SysFileWrite(hFile, ADR(pos), SIZEOF(pos));
	SysFileWrite(hFile, ADR(Logger.TLen), SIZEOF(Logger.TLen));
	SysFileClose(hFile);
END_IF
END_FUNCTION

(* POU Utils Functions/MEMCPY, ST *)
FUNCTION MEMCPY:BOOL
VAR_INPUT
	pSourceAddress:POINTER TO ARRAY[1..2] OF BYTE;
	pDestinationAddress:POINTER TO ARRAY[1..2] OF BYTE;
	BytesToCopy:WORD;
END_VAR
VAR
END_VAR
WHILE (BytesToCopy > 0) DO
	pDestinationAddress^[1]:=pSourceAddress^[1]; (* copy bytes from source to destination *)
	pDestinationAddress:=ADR(pDestinationAddress^[2]); (* increment destination *)
	pSourceAddress:=ADR(pSourceAddress^[2]);(* increment source *)
	BytesToCopy:=BytesToCopy -1; (* decrement number of bytes to copy *)
END_WHILE
END_FUNCTION

(* POU Plant/SYS_Proc, ST *)
PROGRAM SYS_Proc
VAR
	fALARM_PB		:FLT_TAP;
(*	fALARM_TB		:FLT_TAP;
	fALARM_PM		:FLT_TAP;	*)

(*	fGZB_ST			:FLT_TAP;  (* GATEWAY ZIGBEE *)*)
(*	fVPN_ST1		:FLT_TAP;  (* VPN CONNECT *)*)
	fVPN_ST2		:FLT_TAP;  (* VPN STATUS *)
(*	fKEY_CT_ST		:FLT_TAP;  (* DOOR1 *)*)
(*	fKEY_SCT_ST		:FLT_TAP;  (* DOOR2 *)*)
	fKEY_QE_ST		:FLT_TAP;  (* DOOR3 *)

END_VAR
(*************** ISPESL *****************)

fALARM_PB(IN:=ALARM_PB);
IF fALARM_PB.EVH THEN
	LogEv(EL_AlarmStop,EO_PBV,1,1,'Over_Pressure_Alarm');
END_IF
(*
fALARM_TB(IN:=ALARM_TB);
IF fALARM_TB.EVH THEN
	LogEv(EL_AlarmStop,EO_TBV,1,1,'Over_Temperature_Alarm');
END_IF

fALARM_PM(IN:=ALARM_PM);
IF fALARM_PM.EVH THEN
	LogEv(EL_AlarmStop,EO_PMV,1,1,'Under_Pressure_Alarm');
END_IF
*)
(****************************************)

(*### VPN Connection Check ###*)(*
fVPN_ST1(IN:=VPN_ST1);
IF fVPN_ST1.EVH THEN
	LogEv(EL_Log,EO_VPN,1,1,'CONNECT_ON');
END_IF
IF fVPN_ST1.EVL THEN
	LogEv(EL_Log,EO_VPN,1,2,'CONNECT_OFF');
END_IF*)

(*### VPN Status Check ###*)
fVPN_ST2(IN:=VPN_ST2);
IF fVPN_ST2.EVH THEN
	LogEv(EL_Log,EO_VPN,1,3,'STATUS_UP');
END_IF
IF fVPN_ST2.EVL THEN
	LogEv(EL_Wrn,EO_VPN,1,4,'STATUS_DOWN');
END_IF

(*### DOOR01 Status Check ###*)(*
fKEY_CT_ST(IN:=KEY_CT_ST);
IF fKEY_CT_ST.EVH THEN
	LogEv(EL_Log,EO_DOOR,1,2,'Centrale_termica_Close');
END_IF
IF fKEY_CT_ST.EVL THEN
	LogEv(EL_Wrn,EO_DOOR,1,1,'Centrale_termica_Open');
END_IF*)

(*### DOOR02 Status Check ###*)(*
fKEY_SCT_ST(IN:=KEY_SCT_ST);
IF fKEY_SCT_ST.EVH THEN
	LogEv(EL_Log,EO_DOOR,2,2,'Sottocentrale_termica_Close');
END_IF
IF fKEY_SCT_ST.EVL THEN
	LogEv(EL_Wrn,EO_DOOR,2,1,'Sottocentrale_termica_Open');
END_IF*)

(*### DOOR03 Status Check ###*)
fKEY_QE_ST(IN:=KEY_QE_ST);
IF fKEY_QE_ST.EVH THEN
	LogEv(EL_Log,EO_DOOR,3,2,'Quadro_Close');
END_IF
IF fKEY_QE_ST.EVL THEN
	LogEv(EL_Wrn,EO_DOOR,3,1,'Quadro_Open');
END_IF
END_PROGRAM

(* POU Utils Functions/AVERAGE_DINT, ST *)
FUNCTION_BLOCK AVERAGE_DINT
VAR_INPUT
	IN: 	DINT;
END_VAR
VAR_OUTPUT
	HI:		DINT;
	AVG:	DINT;
	LOW:	DINT;
	ERR:	BOOL;
END_VAR
VAR
	sum:	REAL;
	cnt:	WORD;
END_VAR
IF cnt>=65000 THEN
	ERR:=TRUE;
	Read();
	sum := sum - DINT_TO_REAL(AVG);
	cnt := cnt - 1;
END_IF

sum := sum + DINT_TO_REAL(IN);
cnt := cnt + 1;

IF IN<LOW THEN LOW:=IN; END_IF
IF IN>HI  THEN HI :=IN; END_IF
END_FUNCTION_BLOCK
ACTION Read:
AVG := REAL_TO_DINT(sum/cnt);
END_ACTION
ACTION Reset:
HI:=IN;
AVG:=IN;
LOW:=IN;
ERR:=FALSE;

sum:=DINT_TO_REAL(IN);
cnt:=1;
END_ACTION

(* POU Utils Functions/AVERAGE_INT, ST *)
FUNCTION_BLOCK AVERAGE_INT
VAR_INPUT
	IN: 	INT;
END_VAR
VAR_OUTPUT
	HI:		INT;
	AVG:	INT;
	LOW:	INT;
	ERR:	BOOL;
END_VAR
VAR
	sum:	DINT;
	cnt:	WORD;
END_VAR
IF cnt>=65000 THEN
	ERR:=TRUE;
	Read();
	sum := sum - AVG;
	cnt := cnt - 1;
END_IF

sum := sum + IN;
cnt := cnt + 1;

IF IN<LOW THEN LOW:=IN; END_IF
IF IN>HI  THEN HI :=IN; END_IF
END_FUNCTION_BLOCK
ACTION Read:
AVG := DINT_TO_INT(sum/cnt);
END_ACTION
ACTION Reset:
HI:=IN;
AVG:=IN;
LOW:=IN;
ERR:=FALSE;

sum:=IN;
cnt:=1;
END_ACTION

(* POU Utils Functions/AVERAGE_T, ST *)
FUNCTION_BLOCK AVERAGE_T
VAR_INPUT
	IN: 	INT;
END_VAR
VAR_OUTPUT
	HI:		INT;
	AVG:	INT;
	LOW:	INT;
	ERR:	BOOL;
END_VAR
VAR
	sum:	DINT;
	cnt:	WORD;
END_VAR
IF cnt>=65000 THEN
	ERR:=TRUE;
	Read();
	sum := sum - AVG;
	cnt := cnt + 1;
END_IF

sum := sum + IN;
cnt := cnt + 1;

IF IN<LOW THEN  LOW:=IN; END_IF
IF IN>HI  THEN HI :=IN; END_IF
END_FUNCTION_BLOCK
ACTION Read:
AVG := DINT_TO_INT(sum/cnt);
END_ACTION
ACTION Reset:
HI:=IN;
AVG:=IN;
LOW:=IN;
ERR:=FALSE;

sum:=IN;
cnt:=1;
END_ACTION

(* POU Utils Functions/BUILD_16TO32, ST *)
FUNCTION BUILD_16TO32 : DWORD
VAR_INPUT
		pSource	:	POINTER TO WORD;
END_VAR
VAR
		Data	:	DWORD;
END_VAR
Data := WORD_TO_DWORD(pSource^);
pSource := pSource + 1;
Data := Data + WORD_TO_DWORD(pSource^) * 65536;

BUILD_16TO32 := Data;
END_FUNCTION

(* POU CLV/CLV__LogEv, ST *)
FUNCTION CLV__LogEv : BOOL
(* === Log error/event ===
   v1.0[27/05/15]
*)
VAR_INPUT
	Level	: en_Logger_ErrLev;
	Object  : en_SYS_Objects;
	Index	: WORD;
	Error	: WORD;
	Message : STRING;
END_VAR
VAR
	s1 : STRING(160);
	i  : INT;
END_VAR
(* Execute error level operations *)
CASE Level OF
	EL_Wrn: 		Sys.Warning:=TRUE;
	EL_Alarm: 		Sys.Alarm  :=TRUE;
	EL_AlarmStop: 	Sys.Alarm  :=TRUE; (* GO TO STOP STATE!! *)
END_CASE

(* Fill lastlog list *)
s1:=CONCAT(Sys.Time_LogString,';Lev=');
s1:=CONCAT(s1,INT_TO_STRING(Level));
s1:=CONCAT(s1,';Obj=');
s1:=CONCAT(s1,INT_TO_STRING(Object));
s1:=CONCAT(s1,';Idx=');
s1:=CONCAT(s1,WORD_TO_STRING(Index));
s1:=CONCAT(s1,';Err=');
s1:=CONCAT(s1,WORD_TO_STRING(Error));
Sys.LastLogs_Dat[Sys.LastLogs_Idx]:=s1;
Sys.LastLogs_Msg[Sys.LastLogs_Idx]:=Message;
Sys.LastLogs_Idx:=Sys.LastLogs_Idx+1;
IF Sys.LastLogs_Idx>5 THEN Sys.LastLogs_Idx:=0; END_IF

(*---------------------------------------------------------------*)
	CLV.LogHead();
(*---------------------------------------------------------------*)

(* Insert ERR *)
s1:=CONCAT('&ERR=',INT_TO_STRING(Level));
s1:=CONCAT(s1,';');
s1:=CONCAT(s1,INT_TO_STRING(Object));
s1:=CONCAT(s1,';');
s1:=CONCAT(s1,WORD_TO_STRING(Index));
s1:=CONCAT(s1,';');
s1:=CONCAT(s1,WORD_TO_STRING(Error));
s1:=CONCAT(s1,';');
ADDSTRING(ADR(Logger.TData), ADR(s1), Logger.TLen);
s1:=Message;
STR_NOSPACES(ADR(s1));
ADDSTRING(ADR(Logger.TData), ADR(s1), Logger.TLen);

(*---------------------------------------------------------------*)
	CLV.LogSend();
(*---------------------------------------------------------------*)
END_FUNCTION

(* POU CLV/CLV_GET_V1, ST *)
FUNCTION_BLOCK CLV_GET_V1
(* === ClevergyAS GET-Protocol ===
   v1.0[21/04/15] - Draft
*)
VAR CONSTANT
	Log_SERVER			: STRING:='';
	Log_IP				: STRING:='192.168.100.3';
	Log_PORT			: WORD  :=80;
	Log_ConnRetries		: BYTE  :=5;
	Log_GETSTART		: STRING:='GET /cygmsrv/hsgm.ashx?';
	Log_GETEND			: STRING:='$R$N$R$N';
	Log_CHECK			: STRING:='True';
	Log_CRLF			: STRING:='$R$N';
	Log_DataFile		: STRING:='S:\LOG.DAT';
	Log_DataFileMaxSize : DWORD :=5000;
	Log_DataFileOldMax	: WORD  :=100;
	Log_DataFileOld		: STRING:='S:\LOG.DAT.zzz';
	Log_IndexFile		: STRING:='S:\LOG.IDX';
	Log_RecoverMsgs		: BYTE  :=25;

	Cmd_PORT			: WORD  :=10;
	Cmd_WELCOME			: STRING:='';

 	tcpc_S_UNKNOWN: BYTE:=0;
END_VAR
VAR_INPUT

	TData		: ARRAY [0..MAX_SEND_TCP_CLIENT] OF BYTE;
	TLen		: DINT;

	(* Temporary variables used by objects *)
	s1			: STRING(256);
	i1			: WORD;

END_VAR
VAR_OUTPUT
END_VAR
VAR
	tcpc			: TCPCLIENT;
	tcpc_TxBuf		: ARRAY [0..MAX_RECEIVE_TCP_CLIENT] OF BYTE;
	tcpc_TxTrig		: BOOL;
	tcpc_RxBuf		: ARRAY [0..MAX_RECEIVE_TCP_CLIENT] OF BYTE;
	tcpc_RxCnt		: DINT;

	tcpc_St			: BYTE; (* Client status *)
	tcpc_SendReq	: BOOL;

	tcps			: TCPSERVER;
	tcps_TxBuf		: ARRAY [0..MAX_RECEIVE_TCP_CLIENT] OF BYTE;
	tcps_TxTrig		: BOOL;
	tcps_RxBuf		: ARRAY [0..MAX_RECEIVE_TCP_CLIENT] OF BYTE;
	tcps_RxCnt		: DINT;

	tcps_St			: BYTE; (* Server status *)

(****************OLD******************)

	LastIdxPos	: DWORD;

(*	tcpc_Open:    	BOOL;
	IpAddr:			DWORD;
	InetAddr:		DWORD;
	Connected:  	BOOL;
	Error:      	DINT; *)

	SendIdx		: DWORD;
	SendLen		: DINT;

	Retry:			BYTE;	(* Counter for connection retries *)
	Recovered:		BYTE;	(* Counter for recovered unsent messages *)

	i:				DINT;
	pos:			DWORD;
	t:				DWORD;
	hFile:			DWORD;
	fn:				STRING;

	(* Command interpreter *)

	Cmd_Buf_U16:	POINTER TO WORD;
	Cmd_Buf_INT:	POINTER TO INT;
	Cmd_BufLen:		WORD;
	Cmd_St:			WORD;

	Cmd_Obj:		WORD;
	Cmd_ObjIdx:		WORD;
	Cmd_C:			WORD;
	Cmd_R:			WORD;
	Cmd_CLen:		WORD;
	Cmd_RLen:		WORD;

	i : WORD;
	j : INT;
	s2 : STRING;

END_VAR
(*=== Execute state machines ===*)
TcpClient();
TcpServer();

(*=== Execute TCP libraries ===*)
tcpc( xStartSend:=tcpc_Send, aReceiveBuffer:=tcpc_RxBuf, diReceiveCount:=tcpc_RxCnt );
tcps( xStartSend:=tcps_Send, aReceiveBuffer:=tcps_RxBuf, diReceiveCount:=tcps_RxCnt );
END_FUNCTION_BLOCK
ACTION LogHead:
TLen:=0;
(* Set GET header *)
ADDSTRING(ADR(TData), ADR(Logger_GETSTART), TLen);

(* Insert Header *)
s1:=INSERT('ID=&V=1&D=',DWORD_TO_STRING(Plant_SN),3);
s1:=CONCAT(s1,Sys.Time_LogString);
s1:=CONCAT(s1,'&S=');
IF Sys.Alarm THEN i:=2; ELSIF Sys.Warning THEN i:=1; ELSE i:=0; END_IF
s1:=CONCAT(s1,BYTE_TO_STRING(i));
ADDSTRING(ADR(TData), ADR(s1), TLen);
END_ACTION
ACTION LogSend:
(* Finalize string *)
ADDSTRING(ADR(Logger.TData), ADR(Logger_GETEND), Logger.TLen);

(* Read log position *)
pos:=SysFileGetSize(Logger_DataFile);
(* Check log size, bckup and erase if no pending messages *)
IF pos>Log_DataFileMaxSize THEN
	t:=SysFileGetSize(Logger_IndexFile,'r');
	IF t=0 THEN
		FOR i:=0 TO Log_DataFileOldMax DO
			fn:=
		END_FOR

		SysFileDelete(Logger_DataFileOld);
		SysFileRename(Logger_DataFile,Logger_DataFileOld);
		pos:=0;
	END_IF
END_IF
(* Write message on log file *)
hFile:=SysFileOpen(Logger_DataFile,'a');
IF hFile<>0 THEN
	SysFileWrite(hFile, ADR(Logger.TData), Logger.TLen);
	SysFileClose(hFile);
ELSE
	Sys.Warning:=TRUE;
END_IF


(* Check logger status *)
IF Logger.SendReq=FALSE THEN
	(* Set log position for recovery *)
	Logger.SendIdx:=pos;
	(* Copy message data *)
	MEMCPY(ADR(Logger.TData),ADR(Logger.SendData),DINT_TO_WORD(Logger.TLen));
	Logger.SendLen:=Logger.TLen;
	(* Trigger request *)
	Logger.SendReq:=TRUE;
ELSE
	(* Add message position+size in recovery indexes *)
	hFile:=SysFileOpen(Logger_IndexFile,'a');
	SysFileWrite(hFile, ADR(pos), SIZEOF(pos));
	SysFileWrite(hFile, ADR(Logger.TLen), SIZEOF(Logger.TLen));
	SysFileClose(hFile);
END_IF
END_ACTION
ACTION MsgChk:
(* Open index file *)
hFile:=SysFileOpen(Logger_IndexFile,'r');
IF hFile=0 THEN
	RETURN;
END_IF
(* Search oldest message to recover *)
SysFileSetPos(hFile,Logger.LastIdxPos);
Logger.SendLen:=0;
REPEAT
	SysFileRead(hFile, ADR(Logger.SendIdx), SIZEOF(Logger.SendIdx));
	pos:=SysFileGetPos(hFile);
	SysFileRead(hFile, ADR(Logger.SendLen), SIZEOF(Logger.SendLen));
UNTIL
	SysFileEOF(hFile) OR Logger.SendLen<>0
END_REPEAT
SysFileClose(hFile);
(* Delete index file when all messages are recovered *)
IF Logger.SendLen=0 THEN
	Logger.LastIdxPos:=0;
	SysFileDelete(Logger_IndexFile);
	RETURN;
END_IF
(* Recover message data *)
hFile:=SysFileOpen(Logger_DataFile,'r');
IF hFile<>0 THEN
	SysFileSetPos(hFile,Logger.SendIdx);
	SysFileRead(hFile,ADR(Logger.SendData),Logger.SendLen);
	Logger.SendReq:=TRUE;
	SysFileClose(hFile);
END_IF
(* Clear index entry *)
hFile:=SysFileOpen(Logger_IndexFile,'a');
IF hFile<>0 THEN
	SysFileSetPos(hFile,pos);
	i:=0;
	SysFileWrite(hFile, ADR(i), 4);
	Logger.LastIdxPos:=SysFileGetPos(hFile);
	SysFileClose(hFile);
END_IF
END_ACTION
ACTION MsgSave:
(* Add log position in recovery indexes *)
hFile:=SysFileOpen(Logger_IndexFile,'a');
SysFileWrite(hFile, ADR(Logger.SendIdx), SIZEOF(Logger.SendIdx));
SysFileWrite(hFile, ADR(Logger.SendLen), SIZEOF(Logger.SendLen));
SysFileClose(hFile);
END_ACTION
ACTION TcpClient:
(*=== State machine ===*)
CASE tcpc_St OF

	S_Logger_UNKNOWN:
		(* Startup *)
		Logger.SendReq:=FALSE;
		Open:=FALSE;
		Logger.Status:=S_Logger_IDLE;

	S_Logger_IDLE:
		(* Wait request *)
		IF Logger.SendReq THEN
			(* Resolve server name or use static IP *)
			IF LEN(Logger_SERVER)=0 THEN
				InetAddr:=SysSockInetAddr(Logger_IP);
			ELSE
				IpAddr:=SysSockGetHostByName(ADR(Logger_SERVER));
				DWORDSWAP(pIn:=ADR(IpAddr), pOut:=ADR(InetAddr));
			END_IF
			TxTrig:=FALSE;
			RxLen:=0;
			(* Open connection *)
			Open:=TRUE;
			Logger.Status:=S_Logger_WAITCONN;
		END_IF

	S_Logger_WAITCONN:
		(* Wait connection *)
		IF Connected THEN
			(* Send data *)
			TxTrig:=TRUE;
			Logger.Status:=S_Logger_WAITTX;
		END_IF
		IF Error>0 THEN
			Open:=FALSE;
			Logger.Status:=S_Logger_ERROR;
		END_IF

	S_Logger_WAITTX:
		(* Wait transmission *)
		IF NOT TxTrig THEN
			Logger.Status:=S_Logger_WAITRESP;
		END_IF
		IF Error>0 THEN
			Open:=FALSE;
			Logger.Status:=S_Logger_ERROR;
		END_IF

	S_Logger_WAITRESP:
		(* Wait response *)
		IF Connected=FALSE (* OR TIMEOUT!! *) THEN
			Open:=FALSE;
			(* Check response *)
			IF RxLen>=4 AND CHKSTRING(pString:=ADR(RxData), pPattern:=ADR(Logger_CHECK)) THEN
				Logger.SendReq:=FALSE;
				Retry:=0;
				(* Check unsent messages to flush *)
				IF Recovered<Logger_RecoverMsgs THEN
					MsgChk();
					IF Logger.SendReq=TRUE THEN
						Recovered:=Recovered+1;
					ELSE
						Recovered:=0;
					END_IF
				ELSE
					Recovered:=0;
				END_IF
				Logger.Status:=S_Logger_IDLE;
			ELSE
				Logger.Status:=S_Logger_ERROR;
			END_IF
		END_IF

	S_Logger_ERROR:
		(* Connection error or send failure *)
		Retry:=Retry+1;
		IF Retry>Logger_ConnRetries THEN
			(* Save message as unsent *)
			MsgSave();
			Logger.SendReq:=FALSE;
			Retry:=0;
		END_IF
		Logger.Status:=S_Logger_IDLE;

ELSE
	Logger.Status:=S_Logger_UNKNOWN;
END_CASE



(*=== Process Rx data ===*)
(*IF RxLen>0 THEN
	RxLen:=0;
END_IF*)
END_ACTION
ACTION TcpServer:
(*=== State machine ===*)
CASE Status OF
	0: (* Startup *)
		TxLen:=0; TxTrig:=FALSE;
		RxLen:=0;
		Enable:=TRUE;
		Status:=1;

	1: (* Wait incoming connection *)
		IF Connected THEN
			(* Log access *)
			LogEv(EL_Log,EO_VPN,1,5,'Remote');
			(* Send welcome message *)
			(*ADDSTRING(pTxData:=ADR(TxData), pString:=ADR(Remote_WELCOME), TxLen:=TxLen);
			TxTrig:=TRUE;*)
			(* Reset vars *)
			Cmd_BufLen:=0;
			Cmd_St:=0;
			Status:=2;
		END_IF
		IF Error>1 THEN
			Enable:=FALSE;
			Status:=0;
		END_IF

	2: (* Wait command *)
		IF RxLen>0 THEN
			(*=== Interpreter start ===*)
			IF Cmd_BufLen+(RxLen/2)>=MAX_RECEIVE_TCP_SERVER THEN
				(* ERROR *)
				Cmd_BufLen:=0;
			ELSE
				i:=HEXTORAW(pString:=ADR(RxData), StringLen:=DINT_TO_WORD(RxLen), pData:=ADR(Cmd_Buf[Cmd_BufLen]));
				Cmd_BufLen:=Cmd_BufLen+i;
			END_IF
			IF Cmd_BufLen>=8 THEN
				Cmd_Buf_U16:=ADR(Cmd_Buf[6]);
				IF Cmd_BufLen>=(8+Cmd_Buf_U16^) THEN
					Cmd_CLen:=Cmd_Buf_U16^;
					Cmd_Buf_U16:=ADR(Cmd_Buf[0]); Cmd_Obj:=Cmd_Buf_U16^;
					Cmd_Buf_U16:=ADR(Cmd_Buf[2]); Cmd_ObjIdx:=Cmd_Buf_U16^;
					Cmd_Buf_U16:=ADR(Cmd_Buf[4]); Cmd_C:=Cmd_Buf_U16^;
					(* Log command *)
					s2:='RCmd_';		s2:=CONCAT(s2,WORD_TO_STRING(Cmd_Obj));
					s2:=CONCAT(s2,'_'); s2:=CONCAT(s2,WORD_TO_STRING(Cmd_ObjIdx));
					s2:=CONCAT(s2,'_'); s2:=CONCAT(s2,WORD_TO_STRING(Cmd_C));
					s2:=CONCAT(s2,'_');	s2:=CONCAT(s2,WORD_TO_STRING(Cmd_CLen));
					LogEv(EL_Log,EO_VPN,1,6,s2);
					(* Execute command *)
					Command();
					Cmd_BufLen:=0;
				END_IF
			END_IF
			(*=== Interpreter end ===*)
			RxLen:=0;
		END_IF
		IF NOT Connected THEN
			Status:=0;
		END_IF

ELSE
	Status:=0;
END_CASE
END_ACTION

(* POU CLV/CLV_POST_V0, ST *)
FUNCTION_BLOCK CLV_POST_V0
VAR_INPUT
END_VAR
VAR_OUTPUT
END_VAR
VAR
END_VAR

END_FUNCTION_BLOCK

(* POU CLV/CLV_SOCK_V0, ST *)
FUNCTION_BLOCK CLV_SOCK_V0
VAR_INPUT
END_VAR
VAR_OUTPUT
END_VAR
VAR
END_VAR

END_FUNCTION_BLOCK

(* POU Utils Functions/COPY_32SWAP16, ST *)
FUNCTION COPY_32SWAP16:BOOL
VAR_INPUT
	pSourceAddress		:POINTER TO ARRAY[1..2] OF WORD;
	pDestinationAddress	:POINTER TO ARRAY[1..2] OF WORD;
END_VAR
VAR
END_VAR
pDestinationAddress^[1]:=pSourceAddress^[2];
pDestinationAddress^[2]:=pSourceAddress^[1];
END_FUNCTION

(* POU LON/Shared/Type scaling functions/FbDecodeSnvtSwitch, ST *)
FUNCTION_BLOCK FbDecodeSnvtSwitch
VAR_INPUT
	value : typSnvtSwitch;
END_VAR
VAR_OUTPUT
	rValue : REAL;
	xState : BOOL;
END_VAR
VAR
END_VAR
rValue := BYTE_TO_REAL(value.bValue) / 2;
xState := (value.siState > 0);
END_FUNCTION_BLOCK

(* POU LON/Shared/Type scaling functions/FbDecodeSnvtTempP, ST *)
FUNCTION_BLOCK FbDecodeSnvtTempP
VAR_INPUT
	value : typSnvtTempP;
END_VAR
VAR_OUTPUT
	rScaledValue : REAL;
END_VAR
VAR
END_VAR
rScaledValue := INT_TO_REAL(value.iSnvtTempP) / 100;
END_FUNCTION_BLOCK

(* POU Utils Functions/FLT_EVENT, ST *)
FUNCTION_BLOCK FLT_EVENT
VAR_INPUT
	IN		: BOOL;
	INITEV	: BOOL:=TRUE;
END_VAR
VAR_OUTPUT
	EVH		: BOOL;
	EVL		: BOOL;
END_VAR
VAR
	init	: BOOL:=FALSE;
	old		: BOOL;
END_VAR
EVH:=FALSE;
EVL:=FALSE;

IF NOT init THEN
	init:=TRUE;
	IF INITEV THEN
		old := NOT IN;
	ELSE
		old := IN;
	END_IF
END_IF

IF old<>IN THEN
	old:=IN;
	IF IN THEN EVH:=TRUE; ELSE EVL:=TRUE; END_IF
END_IF
END_FUNCTION_BLOCK

(* POU Utils Functions/FLT_TIME, ST *)
FUNCTION_BLOCK FLT_TIME
VAR_INPUT
	IN		: BOOL;
	TTAP	: TIME:=T#5s;
	INITEV	: BOOL:=TRUE;
END_VAR
VAR_OUTPUT
	OUT		: BOOL;
	EVH		: BOOL;
	EVL		: BOOL;
END_VAR
VAR
	init	: BOOL:=FALSE;
	timer	: TON;
END_VAR
EVH:=FALSE;
EVL:=FALSE;

IF NOT init THEN
	init := TRUE;
	IF INITEV THEN
		OUT  := NOT IN;
	ELSE
		OUT  := IN;
	END_IF
END_IF

IF OUT<>IN THEN
	timer(IN:=TRUE,PT:=TTAP);
	IF timer.Q THEN
		OUT:=IN;
		timer(IN:=FALSE);
		IF OUT THEN EVH:=TRUE; ELSE EVL:=TRUE; END_IF
	END_IF
ELSE
	timer(IN:=FALSE);
END_IF
END_FUNCTION_BLOCK

(* POU LON/Module_1/Internal/FuDoCpUpdate_Module_1, ST *)
FUNCTION FuDoCpUpdate_Module_1 : BOOL
(******************************************)
(* Automatic generated code, do not edit! *)
(******************************************)
VAR_INPUT
	ptCp : POINTER TO BYTE;
	ptCpLast : POINTER TO BYTE;
	wCpIndex : WORD;
	uiCpLength : UINT;
	uiCpVariableLength : UINT;
END_VAR
OutDataTelegram_Module_1[0] := C2M_CP_VALUE;
OutDataTelegram_Module_1[1] := WORD_TO_BYTE(wCpIndex AND 16#FF);
OutDataTelegram_Module_1[2] := WORD_TO_BYTE((wCpIndex / 256) AND 16#FF);

mbxModule_1.bTxPrio := 1;
mbxModule_1.bTxProtID := 0;
mbxModule_1.pbTxData := ADR(OutDataTelegram_Module_1);
mbxModule_1.unTxLen := 3 + uiCpLength;
mbxModule_1.MBX_SEND();

IF (mbxModule_1.nError <> MBX_OK) THEN
	FuDoCpUpdate_Module_1 := FALSE;
	RETURN;
END_IF

FuMemCopy(ptCp, ptCpLast, uiCpVariableLength);

FuDoCpUpdate_Module_1 := TRUE;
END_FUNCTION

(* POU LON/Shared/Type scaling functions/FuEncodeSnvtSwitch, ST *)
FUNCTION FuEncodeSnvtSwitch : typSnvtSwitch
VAR_INPUT
	rValue : REAL;
	xState : BOOL;
END_VAR
VAR
END_VAR
IF rValue < 0 THEN rValue := 0; END_IF
IF rValue > 100 THEN rValue := 100; END_IF
FuEncodeSnvtSwitch.bValue := REAL_TO_BYTE(rValue * 2);
IF xState THEN
	FuEncodeSnvtSwitch.siState := 1;
ELSE
	FuEncodeSnvtSwitch.siState := 0;
END_IF
END_FUNCTION

(* POU LON/Shared/Type scaling functions/FuEncodeSnvtTempP, ST *)
FUNCTION FuEncodeSnvtTempP : typSnvtTempP
VAR_INPUT
	rValue : REAL;
END_VAR
VAR
END_VAR
IF rValue < -273.17 THEN rValue := -273.17; END_IF
IF rValue > 327.66 THEN rValue := 327.66; END_IF
FuEncodeSnvtTempP.iSnvtTempP := REAL_TO_INT(rValue * 100);
END_FUNCTION

(* POU LON/Shared/Internal/FuRawToSnvtAlarm, ST *)
FUNCTION FuRawToSnvtAlarm : BOOL
(******************************************)
(* Automatic generated code, do not edit! *)
(******************************************)
VAR_INPUT
	RawDataIn : POINTER TO ARRAY[0..28] OF BYTE;
	DataOut : POINTER TO typSnvtAlarm;
END_VAR
VAR
END_VAR
DataOut^.abLocation[0] := RawDataIn^[0];
DataOut^.abLocation[1] := RawDataIn^[1];
DataOut^.abLocation[2] := RawDataIn^[2];
DataOut^.abLocation[3] := RawDataIn^[3];
DataOut^.abLocation[4] := RawDataIn^[4];
DataOut^.abLocation[5] := RawDataIn^[5];

DataOut^.wObjectId := RawDataIn^[6] * 256 + RawDataIn^[7];

DataOut^.bAlarmType := RawDataIn^[8];

DataOut^.bPriorityLevel := RawDataIn^[9];

DataOut^.wIndexToSnvt := RawDataIn^[10] * 256 + RawDataIn^[11];

DataOut^.abValue[0] := RawDataIn^[12];
DataOut^.abValue[1] := RawDataIn^[13];
DataOut^.abValue[2] := RawDataIn^[14];
DataOut^.abValue[3] := RawDataIn^[15];

DataOut^.wYear := RawDataIn^[16] * 256 + RawDataIn^[17];

DataOut^.bMonth := RawDataIn^[18];

DataOut^.bDay := RawDataIn^[19];

DataOut^.bHour := RawDataIn^[20];

DataOut^.bMinute := RawDataIn^[21];

DataOut^.bSecond := RawDataIn^[22];

DataOut^.wMillisecond := RawDataIn^[23] * 256 + RawDataIn^[24];

DataOut^.abAlarmLimit[0] := RawDataIn^[25];
DataOut^.abAlarmLimit[1] := RawDataIn^[26];
DataOut^.abAlarmLimit[2] := RawDataIn^[27];
DataOut^.abAlarmLimit[3] := RawDataIn^[28];

FuRawToSnvtAlarm := TRUE;
END_FUNCTION

(* POU LON/Shared/Internal/FuRawToSnvtFilePos, ST *)
FUNCTION FuRawToSnvtFilePos : BOOL
(******************************************)
(* Automatic generated code, do not edit! *)
(******************************************)
VAR_INPUT
	RawDataIn : POINTER TO ARRAY[0..5] OF BYTE;
	DataOut : POINTER TO typSnvtFilePos;
END_VAR
VAR
END_VAR
DataOut^.diRwPtr := RawDataIn^[0] * 16777216 + RawDataIn^[1] * 65536 + RawDataIn^[2] * 256 + RawDataIn^[3];

DataOut^.wRwLength := RawDataIn^[4] * 256 + RawDataIn^[5];

FuRawToSnvtFilePos := TRUE;
END_FUNCTION

(* POU LON/Shared/Internal/FuRawToSnvtFileReq, ST *)
FUNCTION FuRawToSnvtFileReq : BOOL
(******************************************)
(* Automatic generated code, do not edit! *)
(******************************************)
VAR_INPUT
	RawDataIn : POINTER TO ARRAY[0..11] OF BYTE;
	DataOut : POINTER TO typSnvtFileReq;
END_VAR
VAR
END_VAR
DataOut^.bRequest := RawDataIn^[0];

DataOut^.wIndex := RawDataIn^[1] * 256 + RawDataIn^[2];

DataOut^.wReceiveTimeout := RawDataIn^[3] * 256 + RawDataIn^[4];

DataOut^.abDestAddress[0] := RawDataIn^[5];
DataOut^.abDestAddress[1] := RawDataIn^[6];
DataOut^.abDestAddress[2] := RawDataIn^[7];
DataOut^.abDestAddress[3] := RawDataIn^[8];
DataOut^.abDestAddress[4] := RawDataIn^[9];

DataOut^.bAuthOn := RawDataIn^[10];

DataOut^.bPrioOn := RawDataIn^[11];

FuRawToSnvtFileReq := TRUE;
END_FUNCTION

(* POU LON/Shared/Internal/FuRawToSnvtFileStatus, ST *)
FUNCTION FuRawToSnvtFileStatus : BOOL
(******************************************)
(* Automatic generated code, do not edit! *)
(******************************************)
VAR_INPUT
	RawDataIn : POINTER TO ARRAY[0..26] OF BYTE;
	DataOut : POINTER TO typSnvtFileStatus;
END_VAR
VAR
END_VAR
DataOut^.bStatus := RawDataIn^[0];

DataOut^.wNumberOfFiles := RawDataIn^[1] * 256 + RawDataIn^[2];

DataOut^.wSelectedFile := RawDataIn^[3] * 256 + RawDataIn^[4];

DataOut^.abAdr[0] := RawDataIn^[5];
DataOut^.abAdr[1] := RawDataIn^[6];
DataOut^.abAdr[2] := RawDataIn^[7];
DataOut^.abAdr[3] := RawDataIn^[8];
DataOut^.abAdr[4] := RawDataIn^[9];
DataOut^.abAdr[5] := RawDataIn^[10];
DataOut^.abAdr[6] := RawDataIn^[11];
DataOut^.abAdr[7] := RawDataIn^[12];
DataOut^.abAdr[8] := RawDataIn^[13];
DataOut^.abAdr[9] := RawDataIn^[14];
DataOut^.abAdr[10] := RawDataIn^[15];
DataOut^.abAdr[11] := RawDataIn^[16];
DataOut^.abAdr[12] := RawDataIn^[17];
DataOut^.abAdr[13] := RawDataIn^[18];
DataOut^.abAdr[14] := RawDataIn^[19];
DataOut^.abAdr[15] := RawDataIn^[20];
DataOut^.abAdr[16] := RawDataIn^[21];
DataOut^.abAdr[17] := RawDataIn^[22];
DataOut^.abAdr[18] := RawDataIn^[23];
DataOut^.abAdr[19] := RawDataIn^[24];
DataOut^.abAdr[20] := RawDataIn^[25];
DataOut^.abAdr[21] := RawDataIn^[26];

FuRawToSnvtFileStatus := TRUE;
END_FUNCTION

(* POU LON/Shared/Internal/FuRawToSnvtHvacMode, ST *)
FUNCTION FuRawToSnvtHvacMode : BOOL
(******************************************)
(* Automatic generated code, do not edit! *)
(******************************************)
VAR_INPUT
	RawDataIn : POINTER TO ARRAY[0..0] OF BYTE;
	DataOut : POINTER TO typSnvtHvacMode;
END_VAR
VAR
END_VAR
DataOut^.bSnvtHvacMode := RawDataIn^[0];

FuRawToSnvtHvacMode := TRUE;
END_FUNCTION

(* POU LON/Shared/Internal/FuRawToSnvtObjRequest, ST *)
FUNCTION FuRawToSnvtObjRequest : BOOL
(******************************************)
(* Automatic generated code, do not edit! *)
(******************************************)
VAR_INPUT
	RawDataIn : POINTER TO ARRAY[0..2] OF BYTE;
	DataOut : POINTER TO typSnvtObjRequest;
END_VAR
VAR
END_VAR
DataOut^.wObjectId := RawDataIn^[0] * 256 + RawDataIn^[1];

DataOut^.bObjectRequest := RawDataIn^[2];

FuRawToSnvtObjRequest := TRUE;
END_FUNCTION

(* POU LON/Shared/Internal/FuRawToSnvtObjStatus, ST *)
FUNCTION FuRawToSnvtObjStatus : BOOL
(******************************************)
(* Automatic generated code, do not edit! *)
(******************************************)
VAR_INPUT
	RawDataIn : POINTER TO ARRAY[0..5] OF BYTE;
	DataOut : POINTER TO typSnvtObjStatus;
END_VAR
VAR
END_VAR
DataOut^.wObjectId := RawDataIn^[0] * 256 + RawDataIn^[1];

DataOut^.bBitfieldByteOffset2 := RawDataIn^[2];

DataOut^.bBitfieldByteOffset3 := RawDataIn^[3];

DataOut^.bBitfieldByteOffset4 := RawDataIn^[4];

DataOut^.bBitfieldByteOffset5 := RawDataIn^[5];

FuRawToSnvtObjStatus := TRUE;
END_FUNCTION

(* POU LON/Shared/Internal/FuRawToSnvtState, ST *)
FUNCTION FuRawToSnvtState : BOOL
(******************************************)
(* Automatic generated code, do not edit! *)
(******************************************)
VAR_INPUT
	RawDataIn : POINTER TO ARRAY[0..1] OF BYTE;
	DataOut : POINTER TO typSnvtState;
END_VAR
VAR
END_VAR
DataOut^.bBitfieldByteOffset0 := RawDataIn^[0];

DataOut^.bBitfieldByteOffset1 := RawDataIn^[1];

FuRawToSnvtState := TRUE;
END_FUNCTION

(* POU LON/Shared/Internal/FuRawToSnvtSwitch, ST *)
FUNCTION FuRawToSnvtSwitch : BOOL
(******************************************)
(* Automatic generated code, do not edit! *)
(******************************************)
VAR_INPUT
	RawDataIn : POINTER TO ARRAY[0..1] OF BYTE;
	DataOut : POINTER TO typSnvtSwitch;
END_VAR
VAR
END_VAR
DataOut^.bValue := RawDataIn^[0];

DataOut^.siState := RawDataIn^[1];

FuRawToSnvtSwitch := TRUE;
END_FUNCTION

(* POU LON/Shared/Internal/FuRawToSnvtTempP, ST *)
FUNCTION FuRawToSnvtTempP : BOOL
(******************************************)
(* Automatic generated code, do not edit! *)
(******************************************)
VAR_INPUT
	RawDataIn : POINTER TO ARRAY[0..1] OF BYTE;
	DataOut : POINTER TO typSnvtTempP;
END_VAR
VAR
END_VAR
DataOut^.iSnvtTempP := RawDataIn^[0] * 256 + RawDataIn^[1];

FuRawToSnvtTempP := TRUE;
END_FUNCTION

(* POU LON/Shared/Internal/FuRawToSnvtTimeStamp, ST *)
FUNCTION FuRawToSnvtTimeStamp : BOOL
(******************************************)
(* Automatic generated code, do not edit! *)
(******************************************)
VAR_INPUT
	RawDataIn : POINTER TO ARRAY[0..6] OF BYTE;
	DataOut : POINTER TO typSnvtTimeStamp;
END_VAR
VAR
END_VAR
DataOut^.iYear := RawDataIn^[0] * 256 + RawDataIn^[1];

DataOut^.bMonth := RawDataIn^[2];

DataOut^.bDay := RawDataIn^[3];

DataOut^.bHour := RawDataIn^[4];

DataOut^.bMinute := RawDataIn^[5];

DataOut^.bSecond := RawDataIn^[6];

FuRawToSnvtTimeStamp := TRUE;
END_FUNCTION

(* POU LON/Module_1/Internal/FuSendCpValueReq_Module_1, ST *)
FUNCTION FuSendCpValueReq_Module_1 : BOOL
(******************************************)
(* Automatic generated code, do not edit! *)
(******************************************)
VAR_INPUT
	ptCp : POINTER TO BYTE;
	ptInternalUseOnly : POINTER TO BYTE;
	wCpIndex : WORD;
END_VAR
IF (ptCp <> 0) THEN
	IF ptInternalUseOnly^.0 = TRUE THEN
		OutDataTelegram_Module_1[0] := C2M_CP_VALUE_QRY;
		OutDataTelegram_Module_1[1] := WORD_TO_BYTE(wCpIndex AND 16#FF);
		OutDataTelegram_Module_1[2] := WORD_TO_BYTE((wCpIndex / 256) AND 16#FF);

		mbxModule_1.bTxPrio := 1;
		mbxModule_1.bTxProtID := 0;
		mbxModule_1.pbTxData := ADR(OutDataTelegram_Module_1);
		mbxModule_1.unTxLen := 3;
		mbxModule_1.MBX_SEND();

		IF (mbxModule_1.nError <> MBX_OK) THEN
			FuSendCpValueReq_Module_1 := FALSE;
			RETURN;
		END_IF
		ptInternalUseOnly^.0 := FALSE;
	END_IF
END_IF

FuSendCpValueReq_Module_1 := TRUE;
END_FUNCTION

(* POU LON/Shared/Internal/FuSnvtFilePosToRaw, ST *)
FUNCTION FuSnvtFilePosToRaw : BOOL
(******************************************)
(* Automatic generated code, do not edit! *)
(******************************************)
VAR_INPUT
	NvDataIn :  POINTER TO typSnvtFilePos;
	DataOut : POINTER TO ARRAY[0..5] OF BYTE;
END_VAR
VAR
END_VAR
DataOut^[0] := DINT_TO_BYTE(SHR(NvDataIn^.diRwPtr, 24));
DataOut^[1] := DINT_TO_BYTE(SHR(NvDataIn^.diRwPtr, 16));
DataOut^[2] := DINT_TO_BYTE(SHR(NvDataIn^.diRwPtr, 8));
DataOut^[3] := DINT_TO_BYTE(NvDataIn^.diRwPtr);

DataOut^[4] := WORD_TO_BYTE(SHR(NvDataIn^.wRwLength, 8));
DataOut^[5] := WORD_TO_BYTE(NvDataIn^.wRwLength);

FuSnvtFilePosToRaw := TRUE;
END_FUNCTION

(* POU LON/Shared/Internal/FuSnvtFileReqToRaw, ST *)
FUNCTION FuSnvtFileReqToRaw : BOOL
(******************************************)
(* Automatic generated code, do not edit! *)
(******************************************)
VAR_INPUT
	NvDataIn :  POINTER TO typSnvtFileReq;
	DataOut : POINTER TO ARRAY[0..11] OF BYTE;
END_VAR
VAR
END_VAR
DataOut^[0] := NvDataIn^.bRequest;

DataOut^[1] := WORD_TO_BYTE(SHR(NvDataIn^.wIndex, 8));
DataOut^[2] := WORD_TO_BYTE(NvDataIn^.wIndex);

DataOut^[3] := WORD_TO_BYTE(SHR(NvDataIn^.wReceiveTimeout, 8));
DataOut^[4] := WORD_TO_BYTE(NvDataIn^.wReceiveTimeout);

DataOut^[5] := NvDataIn^.abDestAddress[0];
DataOut^[6] := NvDataIn^.abDestAddress[1];
DataOut^[7] := NvDataIn^.abDestAddress[2];
DataOut^[8] := NvDataIn^.abDestAddress[3];
DataOut^[9] := NvDataIn^.abDestAddress[4];

DataOut^[10] := NvDataIn^.bAuthOn;

DataOut^[11] := NvDataIn^.bPrioOn;

FuSnvtFileReqToRaw := TRUE;
END_FUNCTION

(* POU LON/Shared/Internal/FuSnvtStateToRaw, ST *)
FUNCTION FuSnvtStateToRaw : BOOL
(******************************************)
(* Automatic generated code, do not edit! *)
(******************************************)
VAR_INPUT
	NvDataIn :  POINTER TO typSnvtState;
	DataOut : POINTER TO ARRAY[0..1] OF BYTE;
END_VAR
VAR
END_VAR
DataOut^[0] := NvDataIn^.bBitfieldByteOffset0;

DataOut^[1] := NvDataIn^.bBitfieldByteOffset1;

FuSnvtStateToRaw := TRUE;
END_FUNCTION

(* POU Utils Functions/LINEAR, ST *)
FUNCTION LINEAR : REAL (* Linear interpolation *)
VAR_INPUT
	X_In	: REAL;
	P1_X	: REAL;
	P1_Y	: REAL;
	P2_X	: REAL;
	P2_Y	: REAL;
END_VAR
VAR
END_VAR
LINEAR:=P1_Y+(((P2_Y-P1_Y)*(X_In-P1_X))/(P2_X-P1_X));
END_FUNCTION

(* POU Utils Functions/LINEAR_BAD, ST *)
FUNCTION LINEAR_BAD : INT (* Linear interpolation *)
VAR_INPUT
	PuntoMinX	: INT;
	PuntoMaxX	: INT;
	ValIn		: INT;
	PuntoMinY	: REAL;
	PuntoMaxY	: REAL;
	Decimali	: BYTE;
END_VAR
VAR
	Gain				: REAL;
	PuntoMinX_R			: REAL;
	PuntoMaxX_R			: REAL;
	Linearizzazione_R	: REAL;
END_VAR
PuntoMinX_R:=INT_TO_REAL(PuntoMinX);
PuntoMaxX_R:=INT_TO_REAL(PuntoMaxX);

Gain:=(PuntoMaxX_R-PuntoMinX_R)/(PuntoMaxY-PuntoMinY);	(* Calcolo in guadagno per la linarizzazione *)
Linearizzazione_R:=PuntoMinx+(Gain*(ValIn-PuntoMinY));	(* Ottengo il valore linearizzato *)

LINEAR_BAD:=REAL_TO_INT(Linearizzazione_R*(EXPT(10, Decimali)));  (* Ottengo intero con i decimai voluti *)
END_FUNCTION

(* POU TCP_Logger/LogTrig, ST *)
FUNCTION LogTrig : BOOL
VAR
	s1 : STRING(160);
	i  : BYTE;
END_VAR
VAR_INPUT
END_VAR
(*---------------------------------------------------------------*)
	Logger_Head();
(*---------------------------------------------------------------*)

CTB01.AddLogData(MBUS:=MBUS01);

CIRD01.AddLogData(ModBus:=MODB01);
CIRD02.AddLogData(ModBus:=MODB01);
CIRD03.AddLogData(ModBus:=MODB01);
CIRD04.AddLogData(ModBus:=MODB01);
CIRD05.AddLogData(ModBus:=MODB01);
CIRD06.AddLogData(ModBus:=MODB01);

TPV01.AddLogData();
TPV02.AddLogData();
TPV03.AddLogData();

ZTHL04.AddLogData(ModBus:=MODB02);
ZTHL05.AddLogData(ModBus:=MODB02);
ZTHL06.AddLogData(ModBus:=MODB02);
ZTHL07.AddLogData(ModBus:=MODB02);
ZTHL08.AddLogData(ModBus:=MODB02);
ZTHL09.AddLogData(ModBus:=MODB02);
ZTHL10.AddLogData(ModBus:=MODB02);
ZTHL11.AddLogData(ModBus:=MODB02);

(*---------------------------------------------------------------*)
	Logger_Send();
(*---------------------------------------------------------------*)
END_FUNCTION

(* POU Utils Functions/MEAN_T, ST *)
FUNCTION MEAN_T : INT
VAR_INPUT
		T1		:	INT;
		T2		:	INT;

		THR_L	:	INT;
		THR_H	:	INT;
END_VAR
VAR
		Tmean	:	INT;
END_VAR
IF T1 >= THR_L AND T1 <= THR_H THEN

	IF T2 >= THR_L AND T2 <= THR_H THEN
		Tmean := (T1 + T2)/2;
	ELSE
		Tmean := T1;
	END_IF
ELSE
	IF T2 >= THR_L AND T2 <= THR_H THEN
		Tmean := T2;
	ELSE
		Tmean := 16#7FFF;	(* No valid temperature data has been passed *)
	END_IF
END_IF

MEAN_T := Tmean;
END_FUNCTION

(* POU Utils Functions/MEMCLR, ST *)
FUNCTION MEMCLR:BOOL
VAR_INPUT
	pDestinationAddress:POINTER TO ARRAY[1..2] OF BYTE;
	BytesToClear:WORD;
END_VAR
VAR
END_VAR
WHILE (BytesToClear > 0) DO
	pDestinationAddress^[1]:=0;
	pDestinationAddress:=ADR(pDestinationAddress^[2]); (* increment destination *)
	BytesToClear:=BytesToClear -1; (* decrement number of bytes to copy *)
END_WHILE
END_FUNCTION

(* POU LON/Module_1/ApplicationMessage/Module_1_ApplicationMsgSend, ST *)
FUNCTION_BLOCK Module_1_ApplicationMsgSend
(******************************************)
(* Automatic generated code, do not edit! *)
(******************************************)
VAR_INPUT
	xSend 		  : BOOL;
	abAddress     : ARRAY[0..10] OF BYTE;
	typServiceSend  : ServiceType;
	xPriority : BOOL;
	xAuthentification : BOOL;
	bMsgCodeSend  : BYTE;
	abMsgDataSend : ARRAY[0..47] OF BYTE;
	bLengthSend	  : BYTE;
END_VAR
VAR_OUTPUT
	bSendStatus   : BYTE;
END_VAR
VAR
	bAddressLength : BYTE;
	RtrigSend : R_TRIG;
END_VAR
RtrigSend(CLK:=xSend);
IF RtrigSend.Q AND (xInitRunning_Module_1 = FALSE) AND (mbxModule_1.bStatus.0) THEN
	OutDataTelegram_Module_1[0] := C2M_LON_MSG_SEND;
	OutDataTelegram_Module_1[1] := INT_TO_BYTE(typServiceSend);
	OutDataTelegram_Module_1[1].6 := xAuthentification;
	OutDataTelegram_Module_1[1].7 := xPriority;
	IF (abAddress[0] = 2) THEN
		bAddressLength := 11;
	ELSE
		bAddressLength := 5;
	END_IF
	FuMemCopy(ADR(abAddress), ADR(OutDataTelegram_Module_1[2]), bAddressLength);
	OutDataTelegram_Module_1[2+bAddressLength] := bMsgCodeSend;
	IF bLengthSend > 48 THEN bLengthSend := 48; END_IF;
	FuMemCopy(ADR(abMsgDataSend), ADR(OutDataTelegram_Module_1[2+bAddressLength+1]), bLengthSend);

	mbxModule_1.bTxPrio := BOOL_TO_BYTE(xPriority);
	mbxModule_1.bTxProtID := 0;
	mbxModule_1.pbTxData := ADR(OutDataTelegram_Module_1);
	mbxModule_1.unTxLen := 3 + bAddressLength + bLengthSend;
	mbxModule_1.MBX_SEND();

	IF (mbxModule_1.nError <> MBX_OK) THEN
		bSendStatus := 255;
	ELSE
		bSendStatus := 0;
	END_IF
END_IF
END_FUNCTION_BLOCK

(* POU LON/Module_1/ApplicationMessage/Module_1_ApplicationMsgSendRsp, ST *)
FUNCTION_BLOCK Module_1_ApplicationMsgSendRsp
(******************************************)
(* Automatic generated code, do not edit! *)
(******************************************)
VAR_INPUT
	xSend 	  : BOOL;
	bCorrelator : BYTE;
	bMsgCode  : BYTE;
	abMsgData : ARRAY[0..47] OF BYTE;
	bLength	  : BYTE;
END_VAR
VAR_OUTPUT
	bSendStatus : BYTE;
END_VAR
VAR
	RtrigSend : R_TRIG;
END_VAR
RtrigSend(CLK:=xSend);
IF RtrigSend.Q AND (xInitRunning_Module_1 = FALSE) AND (mbxModule_1.bStatus.0) THEN
	OutDataTelegram_Module_1[0] := C2M_LON_MSG_RSP_SEND;
	OutDataTelegram_Module_1[1] := bCorrelator;
	OutDataTelegram_Module_1[2] := bMsgCode;
	IF bLength > 48 THEN bLength := 48; END_IF;
	FuMemCopy(ADR(abMsgData), ADR(OutDataTelegram_Module_1[3]), bLength);

	mbxModule_1.bTxPrio := BOOL_TO_BYTE(bCorrelator.7);
	mbxModule_1.bTxProtID := 0;
	mbxModule_1.pbTxData := ADR(OutDataTelegram_Module_1);
	mbxModule_1.unTxLen := 3 + bLength;
	mbxModule_1.MBX_SEND();

	IF (mbxModule_1.nError <> MBX_OK) THEN
		bSendStatus := 255;
	ELSE
		bSendStatus := 0;
	END_IF
END_IF
END_FUNCTION_BLOCK

(* POU Utils Functions/MUX_T, ST *)
FUNCTION MUX_T : INT
(* Manage temperatures measured by different probes in the same room/environment, considering possible probe measurement errors *)
VAR_INPUT
	T1		:	INT;
	T2		:	INT;
	T3		:	INT;
	(*T4		:	INT := 0;*)

	Err1	:	BOOL := TRUE;
	Err2	:	BOOL := TRUE;
	Err3	:	BOOL := TRUE;
	(*Err4	:	BOOL := TRUE;*)

	Used	:	BYTE;

END_VAR
VAR
	Sum		:	INT;
	count	:	BYTE;
END_VAR
CASE Used OF

	1:	(* T1 passed *)
		IF Err1 THEN
			Sum := 16#7FFF;
		ELSE
			Sum := T1;
			count := 1;
		END_IF

	2:	(* T1, T2 passed *)
		IF Err1 THEN
			IF Err2 THEN
				Sum := 16#7FFF;
			ELSE
				Sum := T2;
				count := 1;
			END_IF
		ELSE
			IF Err2 THEN
				Sum := T1;
				count := 1;
			ELSE
				Sum := T1 + T2;
				count := 2;
			END_IF
		END_IF

	3:	(* T1, T2, T3 passed *)
		IF Err1 THEN
			IF Err2 THEN
				IF Err3 THEN
					Sum := 16#7FFF;
				ELSE
					Sum := T3;
					count := 1;
				END_IF
			ELSE
				IF Err3 THEN
					Sum := T2;
					count := 1;
				ELSE
					Sum := T2 + T3;
					count := 2;
				END_IF
			END_IF
		ELSE
			IF Err2 THEN
				IF Err3 THEN
					Sum := T1;
					count := 1;
				ELSE
					Sum := T1 + T3;
					count := 2;
				END_IF
			ELSE
				IF Err3 THEN
					Sum := T1 + T2;
					count := 2;
				ELSE
					Sum := T1 + T2 + T3;
					count := 3;
				END_IF
			END_IF
		END_IF
(*
	4:
		IF Err1 THEN
			IF Err2 THEN
				IF Err3 THEN
					IF Err4 THEN
						Sum := 16#7FFF;
					ELSE
						Sum := T4;
						count := 1;
					END_IF
				ELSE
					IF Err4 THEN
						Sum := T3;
						count := 1;
					ELSE
						Sum := T3 + T4;
						count := 2;
					END_IF
				END_IF
			ELSE
				IF Err3 THEN
					IF Err4 THEN
						Sum := T2;
						count := 1;
					ELSE
						Sum := T2 + T4;
						count := 2;
					END_IF
				ELSE
					IF Err4 THEN
						Sum := T2 + T3;
						count := 2;
					ELSE
						Sum := T2 + T3 + T4;
						count := 3;
					END_IF
				END_IF
			END_IF
		ELSE
			IF Err2 THEN
				IF Err3 THEN
					IF Err4 THEN
						Sum := T1;
					ELSE
						Sum := T1 + T4;
						count := 2;
					END_IF
				ELSE
					IF Err4 THEN
						Sum := T1 + T3;
						count := 2;
					ELSE
						Sum := T1 + T3 + T4;
						count := 3;
					END_IF
				END_IF
			ELSE
				IF Err3 THEN
					IF Err4 THEN
						Sum := T1 + T2;
						count := 2;
					ELSE
						Sum := T1 + T2 + T4;
						count := 3;
					END_IF
				ELSE
					IF Err4 THEN
						Sum := T1 + T2 + T3;
						count := 3;
					ELSE
						Sum := T1 + T2 + T3 + T4;
						count := 4;
					END_IF
				END_IF
			END_IF
		END_IF
*)
END_CASE

IF Sum = 16#7FFF THEN
	(* No valid data -> return default *)
	MUX_T := Plant_DefaultTAmb;
ELSE
	(* Do average *)
	MUX_T := Sum/count;
END_IF
END_FUNCTION

(* POU Plant_Objects/obj_CAL_VT100GC1B, ST *)
FUNCTION_BLOCK obj_CAL_VT100GC1B
(* === CALDAIA VIESSMAN via LON ===
   v1.0[16/04/15] - Versioning
*)
VAR_INPUT
	(* Settings *)
	ID				: BYTE;
	(* Controls *)
	Run				: BOOL;

	(* LON Status *)
	ModuleState	  : DWORD;
	(*** LON to CAL ***)
	(* Node inputs *)
	NO_Request    : typSnvtObjRequest;
	NO_TimeSet    : typSnvtTimeStamp;
	NO_AlarmSet   : typSnvtAlarm;
	(* Domestic hot water controller *)
	DHW_ModeSet   : typSnvtHvacMode;
	DHW_SetPoint  : typSnvtTempP;
	(* Central flow demand manager *)
	CFD_SetEnable : typSnvtSwitch;
	CFD_SetMode   : typSnvtHvacMode;
	CFD_SetPoint  : typSnvtTempP;
	(* LON From CAL *)
	NO_Status     : typSnvtObjStatus;
	NO_Alarm      : typSnvtAlarm;
	NO_RlyState   : typSnvtState;
	DHW_ActTemp   : typSnvtTempP;			(* Actual DHW temperature *)
	DHW_SetTemp   : typSnvtTempP;			(* Actual temperature set point *)
	CFD_GetEnable : typSnvtSwitch;
	CFD_Temp      : typSnvtTempP;
	CFD_SetTemp   : typSnvtTempP;

	Temperature	:  	INT;
END_VAR
VAR_IN_OUT
	CLIM		  : typ_Clima;
END_VAR
VAR_OUTPUT
	(* Status *)
	Status_Log	: BYTE;
	Status_Vis 	: DWORD;
END_VAR
VAR
	InitOK		: BOOL;
	fAlarm		: BOOL;
	fAlarmBUS	: BOOL;
	fWarning	: BOOL;

	Curve 		: CHARCURVE;
	Curve_Err 	: BYTE;
	Curve_Temp	: INT;

	Timer1		: TON;		(* Refresh timer for output vars *)

END_VAR
(* Check initialization *)
IF NOT InitOK THEN Init(); END_IF

(* Check LON connection *)
(*
...
*)

(* Check state *)
IF NO_Alarm.bAlarmType=1 THEN
	IF NOT fAlarm THEN
		fAlarm:=TRUE;
		LogEv(EL_Alarm,EO_CAL,ID,4,RAWTOHEXSTR(ADR(NO_Alarm.abAlarmLimit[2]),2));
	END_IF
ELSE
	fAlarm:=FALSE;
END_IF

(* Check climatic setup *)
IF NOT CLIM.InitOK THEN Clima_Default(); END_IF;
(* Calculate Setpoint *)
Curve(	IN:= Temperature,	N:= 5, P:= CLIM.Points,
		OUT=> Curve_Temp, ERR=> Curve_Err );
IF Curve_Err>0 THEN
	IF NOT fWarning THEN
		fWarning:=TRUE;
		LogEv(EL_Wrn,EO_CAL,ID,2,'Climatic_Error');
	END_IF
ELSE
	fWarning:=FALSE;
END_IF

(* Send temperature set-point (force update every 1min) *)
CFD_SetPoint.iSnvtTempP:=Curve_Temp*10;

(* Attivazione caldaia *)
IF Run THEN
	CFD_SetMode.bSnvtHvacMode := 0;		(* Automatic mode *)
ELSE
	CFD_SetMode.bSnvtHvacMode := 3;		(* Off *)
END_IF

(* Status color *)
   IF fAlarm OR fAlarmBUS	THEN Status_Log:=2; Status_Vis:=COLOR_RED;
ELSIF fWarning 		   		THEN Status_Log:=1; Status_Vis:=COLOR_YELLOW;
              				ELSE Status_Log:=0; Status_Vis:=SEL(Run,16#006000,16#20F020);
END_IF

Lamp.obj_Status := Status_Log;
Lamp.UpdateStatus();
END_FUNCTION_BLOCK
ACTION Clima_Default:
CLIM.Points[0].X:=-300; CLIM.Points[0].Y:=650;
CLIM.Points[1].X:=-50 ; CLIM.Points[1].Y:=650;
CLIM.Points[2].X:= 200; CLIM.Points[2].Y:=200;
CLIM.Points[3].X:= 300; CLIM.Points[3].Y:=200;
CLIM.Points[4].X:= 500; CLIM.Points[4].Y:=200;
CLIM.InitOK:=TRUE;
LogEv(EL_Wrn,EO_CAL,ID,1,'Climatic_default');
END_ACTION
ACTION Heartbeat:
(* Call this at same cycle of LON execution call *)
Timer1(IN:=NOT CAL01.Timer1.Q,PT:=T#1m);
CFD_SetPoint.bStatusInformation:=SEL(CAL01.Timer1.Q,0,16#80);		(* Re-trigger transmission every 60s *)
END_ACTION
ACTION Init:
(**** CAL01.CFD_SetEnable.bValue:=0; *)

(*CAL01.CFD_SetEnable.siState:=16#FF; (* Default value: AUTO *)*)

(**** CAL01.CFD_SetMode.bSnvtHvacMode:=16#FF; (* Default value: AUTO *) *)

(*CAL01.CFD_SetPoint.iSnvtTempP:=0; (* Default temperature: 0°C *)*)

(* End initialization *)
InitOK:=TRUE;
END_ACTION

(* POU Utils Functions/RAWTOHEXSTR, ST *)
FUNCTION RAWTOHEXSTR : STRING(128)
VAR_INPUT
	pData: POINTER TO BYTE;
	DataLen: BYTE;
END_VAR
VAR
	pt: POINTER TO BYTE;
	xl: BYTE;
END_VAR
pt:=ADR(RAWTOHEXSTR);

xl:=2;

WHILE DataLen>0 AND xl<128 DO

	pt^ := (pData^ / 16#10) + 48 + (((pData^ / 16#10)/10)*7);
	pt:=pt+1;
	pt^ := (pData^ AND 16#0F)  + 48 + (((pData^ AND 16#0F)/10)*7);
	pt:=pt+1;

	xl:=xl+2;

	DataLen:=DataLen-1;
	pData:=pData+1;

END_WHILE

pt^:=0;
END_FUNCTION

(* POU Plant_Objects/obj_CRON, ST *)
FUNCTION_BLOCK obj_CRON
(* === CRONOGRAFO STANDARD ===
   v1.0[16/04/15] - Versioning
   v1.1[19/05/15] - Removed DB creation from previous year
*)
VAR_INPUT
	(* Settings *)
	ID			: BYTE;		(* Index of instanced object *)

	InitOK		: BOOL;
	Alarm		: BOOL;
	Warning		: BOOL;

	Profile		: typ_Cron_Profile; 				(* Profilo attivo *)
	ProfileNr	: BYTE;								(* Indice profilo attivo *)
	CalendarIdx : WORD;								(* Indice calendario attivo *)
	Jolly		: ARRAY[0..9] OF typ_Cron_Jolly;	(* Jolly attivi *)

END_VAR
VAR_IN_OUT
END_VAR
VAR_OUTPUT
	SetPoint		: INT;
	(* Status *)
	Status_Log		: BYTE;
	Status_Vis 		: DWORD;
END_VAR
VAR
	Buf: 	ARRAY[0..512] OF BYTE; (* AVOID THIS!! *)
	hFile: 	DWORD;
	sFile: 	STRING;
	sFile2: STRING;

	i:		WORD;
	t1:		DWORD;
	t2:		BOOL;

END_VAR
(* Check initialization *)
IF NOT InitOK THEN Init(); END_IF

(* Chrono *)
IF CalendarIdx<>Sys.Time_CT_Day THEN DB_Load(); END_IF
SetPoint:=Profile.Setpoint[Sys.Time_CT_Quarter];

(* Check jolly *)
FOR i := 0 TO 9 DO
	IF ( DT_TO_DWORD(Jolly[i].Start)>0  AND Jolly[i].End>Jolly[i].Start AND
	     Jolly[i].Start<=Sys.Time_CT_DT AND Jolly[i].End>Sys.Time_CT_DT ) THEN
			SetPoint:=Jolly[i].Temp;
	END_IF
END_FOR


(* Status color *)
   IF Alarm   THEN Status_Log:=2; Status_Vis:=COLOR_RED;
ELSIF Warning THEN Status_Log:=1; Status_Vis:=COLOR_YELLOW;
              ELSE Status_Log:=0; Status_Vis:=COLOR_GREEN;
			  END_IF
END_FUNCTION_BLOCK
ACTION DB_Create:
(* Create empty file *)
hFile:=SysFileOpen(FileName:=sFile, Mode:='w');

MEMCLR(pDestinationAddress:=ADR(Buf), BytesToClear:=SIZEOF(Buf));
FOR i := 0 TO 10239 BY 512 DO
	t1:=SysFileWrite(File:=hFile, Buffer:=ADR(Buf), Size:=512);		(* Clear created file (all bytes 0) *)
END_FOR
Buf[0]:=1;
t2:=SysFileSetPos(File:=hFile, Pos:=0);
t1:=SysFileWrite(File:=hFile, Buffer:=ADR(Buf), Size:=1);
SysFileClose(File:=hFile);
END_ACTION
ACTION DB_Load:
DB_SetName();

(* Open data file *)
hFile:=SysFileOpen(FileName:=sFile, Mode:='r');

(* File not found *)
IF hFile=0 THEN
	Warning:=TRUE;
	LogEv(EL_Wrn,EO_CRON,ID,1,'No_data_file');
	DB_Create();
	(* Reopen file *)
	hFile:=SysFileOpen(FileName:=sFile, Mode:='r');
	IF hfile=0 THEN
		Alarm:=TRUE;
		LogEv(EL_Alarm,EO_CRON,ID,3,'Filesystem_error');
		RETURN;
	END_IF
END_IF

(* Check version *)
SysFileRead(File:=hFile, Buffer:=ADR(Buf), Size:=1);
IF Buf[0]<>1 THEN
	IF NOT Alarm THEN
		Alarm:=TRUE;
		LogEv(EL_Alarm,EO_CRON,ID,2,'Bad_data_version');
	END_IF
	SysFileClose(File:=hFile);
	RETURN;
END_IF

(* Read Jolly data *)
t2:=SysFileSetPos(File:=hFile, Pos:=512);
t1:=SysFileRead(File:=hFile, Buffer:=ADR(Jolly), Size:=SIZEOF(Jolly));
(* Read active profile index *)
CalendarIdx:=Sys.Time_CT_Day;
t2:=SysFileSetPos(File:=hFile, Pos:=(1024+4*CalendarIdx));
t1:=SysFileRead(File:=hFile, Buffer:=ADR(ProfileNr), Size:=SIZEOF(ProfileNr));
(* Read active profile *)
t2:=SysFileSetPos(File:=hFile, Pos:=(3072+512*ProfileNr));
t1:=SysFileRead(File:=hFile, Buffer:=ADR(Profile), Size:=SIZEOF(Profile));

(* Close file and validate data *)
SysFileClose(File:=hFile);
END_ACTION
ACTION DB_SetName:
(* Create current filename 'yyyyCRnn.DAT' *)
sFile:=CONCAT(FilesPath,WORD_TO_STRING(Sys.Time_Year));
sFile:=CONCAT(STR1:=sFile, STR2:='CR');
IF ID<10 THEN
sFile:=CONCAT(STR1:=sFile, STR2:='0');
END_IF
sFile:=CONCAT(STR1:=sFile, STR2:=BYTE_TO_STRING(ID));
sFile:=CONCAT(STR1:=sFile, STR2:='.DAT');
END_ACTION
ACTION Init:
DB_Load();
InitOK:=TRUE;
END_ACTION

(* POU Plant_Objects/obj_CRON_EDITOR, ST *)
FUNCTION_BLOCK obj_CRON_EDITOR
(* === EDITOR CRONOGRAFO ===
   v1.0[16/04/15] - Versioning
   v1.1[19/05/15] - Create empty profile when not found
*)
VAR_INPUT

	(* Common selections *)
	CN_Sel:			BYTE:=1;
	CN_Act:			BYTE;
	CN_YSel:		WORD:=2015;
	CN_YAct:		WORD;

	(* Profile editor *)
	PR_Sel: 		BYTE:=1;
	PR_Act:			BYTE;
	PR_TT:			REAL;
	PR:				typ_Cron_Profile;
	(* Profile signals *)
	PR_Load:		BOOL;
	PR_Save:		BOOL;

	(* Calendar editor *)
	CA_Sel:			BYTE:=1; (* Calendar month selected *)
	CA_Act:			BYTE;    (* Calendar month active *)
	CA_DayF:		BYTE:=0;
	CA_DayL:		BYTE:=31;
	CA_TPR:			BYTE;
	CA:				typ_Cron_Calendar; (* Only used for first 32 entries *)
	(* Calendar signals *)
	CA_Load:		BOOL;
	CA_Save:		BOOL;

	(* Jolly editor *)
	JL:				ARRAY[0..9] OF typ_Cron_Jolly;
	(* Jolly signals *)
	JL_Load:		BOOL;
	JL_Save:		BOOL;

END_VAR
VAR_OUTPUT
	Message		: STRING;
END_VAR
VAR
	sFileName	: STRING;
	sFileMode	: STRING;
	hFile		: DWORD;
	Buf			: ARRAY[0..512] OF BYTE; (* AVOID THIS!! *)

	i			: WORD;
	ver			: BYTE;
	r1			: BOOL;
	r2			: DWORD;

END_VAR
IF PR_Load THEN PR_Load_Exe(); PR_Load:=FALSE; END_IF
IF PR_Save THEN PR_Save_Exe(); PR_Save:=FALSE; END_IF
IF CA_Load THEN CA_Load_Exe(); CA_Load:=FALSE; END_IF
IF CA_Save THEN CA_Save_Exe(); CA_Save:=FALSE; END_IF
IF JL_Load THEN JL_Load_Exe(); JL_Load:=FALSE; END_IF
IF JL_Save THEN JL_Save_Exe(); JL_Save:=FALSE; END_IF
END_FUNCTION_BLOCK
ACTION CA_Load_Exe:
sFileMode:='r';
FileOpen();

IF hFile<>0 THEN

	(* Read calendar month *)
	FOR i := 0 TO 31 DO
		r1:=SysFileSetPos(File:=hFile, Pos:=(1024 + ((CA_Sel-1)*32 + i)*4));
		r2:=SysFileRead(File:=hFile, Buffer:=ADR(CA.Profile[i]), Size:=1);
	END_FOR

	(* Close file *)
	SysFileClose(File:=hFile);

	(* Validate data *)
	CA_Act :=CA_Sel;
	CN_Act :=CN_Sel;
	CN_YAct:=CN_YSel;

	Message:='Calendar load OK';

END_IF
END_ACTION
ACTION CA_Save_Exe:
sFileMode:='a';
FileOpen();

IF hFile<>0 THEN

	(* Write calendar month *)
	FOR i := 0 TO 31 DO
		r1:=SysFileSetPos(File:=hFile, Pos:=(1024 + ((CA_Sel-1)*32 + i)*4));
		r2:=SysFileGetPos(hFile);
		r2:=SysFileWrite(File:=hFile, Buffer:=ADR(CA.Profile[i]), Size:=1);
	END_FOR

	(* Close file *)
	SysFileClose(File:=hFile);

	Message:='Calendar save OK';

END_IF
END_ACTION
ACTION FileOpen:
(* Create current filename 'yyyyCRnn.DAT' *)
sFileName:=CONCAT(FilesPath,WORD_TO_STRING(CN_YSel));
sFileName:=CONCAT(STR1:=sFileName, STR2:='CR');
IF CN_Sel<10 THEN
sFileName:=CONCAT(STR1:=sFileName, STR2:='0');
END_IF
sFileName:=CONCAT(STR1:=sFileName, STR2:=BYTE_TO_STRING(CN_Sel));
sFileName:=CONCAT(STR1:=sFileName, STR2:='.DAT');

(* Check file version and size! *)
(* ... *)

(* Open data file *)
hFile:=SysFileOpen(FileName:=sFileName, Mode:='r');

(* File not found *)
IF hFile=0 THEN
	Message:='File not found - created empty file';
	(* Create empty file *)
	hFile:=SysFileOpen(FileName:=sFileName, Mode:='w');
	MEMCLR(pDestinationAddress:=ADR(Buf), BytesToClear:=SIZEOF(Buf));
	FOR i := 0 TO 10239 BY 512 DO
		SysFileWrite(File:=hFile, Buffer:=ADR(Buf), Size:=512);
	END_FOR
	Buf[0]:=1;
	SysFileSetPos(File:=hFile, Pos:=0);
	SysFileWrite(File:=hFile, Buffer:=ADR(Buf), Size:=1);
END_IF

(* Close file *)
SysFileClose(File:=hFile);

(* Open data file *)
hFile:=SysFileOpen(FileName:=sFileName, Mode:=sFileMode);
END_ACTION
ACTION JL_Load_Exe:
sFileMode:='r';
FileOpen();

IF hFile<>0 THEN

	(* Read jolly *)
	r1:=SysFileSetPos(File:=hFile, Pos:=512);
	r2:=SysFileRead(File:=hFile, Buffer:=ADR(JL), Size:=SIZEOF(JL));

	(* Close file *)
	SysFileClose(File:=hFile);

	(* Validate data *)
	CN_Act:=CN_Sel;
	CN_YAct:=CN_YSel;

	Message:='Jolly load OK';

END_IF
END_ACTION
ACTION JL_Save_Exe:
sFileMode:='a';
FileOpen();

IF hFile<>0 THEN

	(* Write selected profile *)
	r1:=SysFileSetPos(File:=hFile, Pos:=512);
	r2:=SysFileWrite(File:=hFile, Buffer:=ADR(JL), Size:=SIZEOF(JL));

	(* Close file *)
	SysFileClose(File:=hFile);

	Message:='Jolly save OK';

END_IF
END_ACTION
ACTION PR_Load_Exe:
sFileMode:='r';
FileOpen();

IF hFile<>0 THEN

	(* Read selected profile *)
	r1:=SysFileSetPos(File:=hFile, Pos:=(3072 + 512*PR_Sel));
	r2:=SysFileRead(File:=hFile, Buffer:=ADR(PR), Size:=SIZEOF(PR));

	(* Close file *)
	SysFileClose(File:=hFile);

	(* Validate data *)
	PR_Act:=PR_Sel;
	CN_Act:=CN_Sel;
	CN_YAct:=CN_YSel;

	Message:='Profile load OK';

END_IF
END_ACTION
ACTION PR_Save_Exe:
sFileMode:='a';
FileOpen();

IF hFile<>0 THEN

	(* Write selected profile *)
	r1:=SysFileSetPos(File:=hFile, Pos:=(3072 + 512*PR_Sel));
	r2:=SysFileWrite(File:=hFile, Buffer:=ADR(PR), Size:=SIZEOF(PR));

	(* Close file *)
	SysFileClose(File:=hFile);

	Message:='Profile save OK';

END_IF
END_ACTION

(* POU Plant_Objects/obj_CRONTER, ST *)
FUNCTION_BLOCK obj_CRONTER
(* === THERMOSTAT ===
   v1.0[30/07/15] - Versioning
*)
VAR CONSTANT
	OFF			: BYTE := 0;
	ON			: BYTE := 1;
	ANTI_FREEZE	: BYTE := 2;
END_VAR
VAR_INPUT
	(* Settings *)
	ID			: BYTE;		(* Index of instanced object *)

	InitOK		: BOOL;
	Alarm		: BOOL;
	Warning		: BOOL;

	Profile		: typ_Cron_Profile; 				(* Profilo attivo *)
	ProfileNr	: BYTE;								(* Indice profilo attivo *)
	CalendarIdx : WORD;								(* Indice calendario attivo *)
	Jolly		: ARRAY[0..9] OF typ_Cron_Jolly;	(* Jolly attivi *)

	Temperature	: INT;
	Local_MaxRunTAmb	:	INT;					(* Local maximum environment temperature, NOT "TAMB" *)

END_VAR
VAR_IN_OUT
END_VAR
VAR_OUTPUT
	SetPoint		: INT;
	Run				: BYTE;

	(* Status *)
	Status_Log		: BYTE;
	Status_Vis 		: DWORD;
END_VAR
VAR
	Buf: 	ARRAY[0..512] OF BYTE; (* AVOID THIS!! *)
	hFile: 	DWORD;
	sFile: 	STRING;
	sFile2: STRING;

	i:		WORD;
	t1:		DWORD;
	t2:		BOOL;

END_VAR
(* Check initialization *)
IF NOT InitOK THEN Init(); END_IF

(* Check Temperature *)
IF Temperature < Local_MaxRunTAmb THEN

	(* LOCAL environment temperature lower than maximum allowed -> Proceed with SetPoint adjustment *)
	(* Chrono *)
	IF CalendarIdx<>Sys.Time_CT_Day THEN DB_Load(); END_IF
	SetPoint:=Profile.Setpoint[Sys.Time_CT_Quarter];

	(* Check jolly *)
	FOR i := 0 TO 9 DO
		IF ( DT_TO_DWORD(Jolly[i].Start)>0  AND Jolly[i].End>Jolly[i].Start AND
		     Jolly[i].Start<=Sys.Time_CT_DT AND Jolly[i].End>Sys.Time_CT_DT ) THEN
				SetPoint:=Jolly[i].Temp;
		END_IF
	END_FOR

	IF SetPoint < 180 THEN
		(* Switch off the device *)
		Run := OFF;
	ELSE
		(* Set according to feedback T - Histeresys of 1°C *)
		IF Temperature >= (SetPoint + 5) THEN
			Run := OFF;
		ELSIF Temperature <= (SetPoint - 5) THEN
			Run := ON;
		END_IF

		(* Between "SetPoint-5" and "SetPoint+5" last state (ON or OFF) of "Run" is kept	*)
	END_IF

ELSE
	(* Environment overtemperature: stop heating -> Stop device *)
	Run := OFF;
END_IF

(* Freeze warning: Switch on and heat! *)
IF Temperature < Plant_AntiFreezeTAmb THEN
	Run := ANTI_FREEZE;
END_IF


(* Status color *)
   IF Alarm   THEN Status_Log:=2; Status_Vis:=COLOR_RED;
ELSIF Warning THEN Status_Log:=1; Status_Vis:=COLOR_YELLOW;
              ELSE Status_Log:=0; Status_Vis:=COLOR_GREEN;
			  END_IF
END_FUNCTION_BLOCK
ACTION DB_Create:
(* Create empty file *)
hFile:=SysFileOpen(FileName:=sFile, Mode:='w');

MEMCLR(pDestinationAddress:=ADR(Buf), BytesToClear:=SIZEOF(Buf));
FOR i := 0 TO 10239 BY 512 DO
	t1:=SysFileWrite(File:=hFile, Buffer:=ADR(Buf), Size:=512);		(* Clear created file (all bytes 0) *)
END_FOR
Buf[0]:=1;
t2:=SysFileSetPos(File:=hFile, Pos:=0);
t1:=SysFileWrite(File:=hFile, Buffer:=ADR(Buf), Size:=1);
SysFileClose(File:=hFile);
END_ACTION
ACTION DB_Load:
DB_SetName();

(* Open data file *)
hFile:=SysFileOpen(FileName:=sFile, Mode:='r');

(* File not found *)
IF hFile=0 THEN
	Warning:=TRUE;
	LogEv(EL_Wrn,EO_CRON,ID,1,'No_data_file');
	DB_Create();
	(* Reopen file *)
	hFile:=SysFileOpen(FileName:=sFile, Mode:='r');
	IF hfile=0 THEN
		Alarm:=TRUE;
		LogEv(EL_Alarm,EO_CRON,ID,3,'Filesystem_error');
		RETURN;
	END_IF
END_IF

(* Check version *)
SysFileRead(File:=hFile, Buffer:=ADR(Buf), Size:=1);
IF Buf[0]<>1 THEN
	IF NOT Alarm THEN
		Alarm:=TRUE;
		LogEv(EL_Alarm,EO_CRON,ID,2,'Bad_data_version');
	END_IF
	SysFileClose(File:=hFile);
	RETURN;
END_IF

(* Read Jolly data *)
t2:=SysFileSetPos(File:=hFile, Pos:=512);
t1:=SysFileRead(File:=hFile, Buffer:=ADR(Jolly), Size:=SIZEOF(Jolly));
(* Read active profile index *)
CalendarIdx:=Sys.Time_CT_Day;
t2:=SysFileSetPos(File:=hFile, Pos:=(1024+4*CalendarIdx));
t1:=SysFileRead(File:=hFile, Buffer:=ADR(ProfileNr), Size:=SIZEOF(ProfileNr));
(* Read active profile *)
t2:=SysFileSetPos(File:=hFile, Pos:=(3072+512*ProfileNr));
t1:=SysFileRead(File:=hFile, Buffer:=ADR(Profile), Size:=SIZEOF(Profile));

(* Close file and validate data *)
SysFileClose(File:=hFile);
END_ACTION
ACTION DB_SetName:
(* Create current filename 'yyyyCRnn.DAT' *)
sFile:=CONCAT(FilesPath,WORD_TO_STRING(Sys.Time_Year));
sFile:=CONCAT(STR1:=sFile, STR2:='CR');
IF ID<10 THEN
sFile:=CONCAT(STR1:=sFile, STR2:='0');
END_IF
sFile:=CONCAT(STR1:=sFile, STR2:=BYTE_TO_STRING(ID));
sFile:=CONCAT(STR1:=sFile, STR2:='.DAT');
END_ACTION
ACTION Init:
DB_Load();
InitOK:=TRUE;
END_ACTION

(* POU Plant_Objects/obj_CTL, ST *)
FUNCTION_BLOCK obj_CTL
(* === PULSE VOLUME COUNTER ===
   v1.0[16/04/15] - Versioning
*)
VAR_INPUT
	(* Settings *)
	ID				: BYTE;	(* Index of instanced object *)
	Peso			: DWORD;
	(* Physical inputs *)
	CTL_ST			: BOOL;
END_VAR
VAR_IN_OUT
	COUNT			: DWORD;
END_VAR
VAR_OUTPUT
	(* Status *)
	Status_Log		: BYTE;
END_VAR
VAR
	Filter			: FLT_TAP := ( INITEV:=FALSE );
	Timer			: TON;
	TCount			: DWORD;
	i				: DWORD;
END_VAR
(* Execute timer *)
Timer(IN:=NOT Timer.Q, PT:=T#60m);

(* Execute filter on counter status *)
Filter(IN:=CTL_ST);

(* Count event *)
IF Filter.EVH THEN
	COUNT:=COUNT+Peso;
	TCount:=TCount+1;
	(* Check flow rate *)
	IF TCount>=Plant_MaxWaterLoss THEN
		i:=(TCount*TIME_TO_DWORD(Timer.PT))/TIME_TO_DWORD(Timer.ET);	(* Estimated mc per hour *)
		i:= i * Peso;

		(* NB The weight is multiplied by 10 -> Need to divide it by 10 server side *)
		LogEv(EL_AlarmStop,EO_CTL,ID,1,DWORD_TO_STRING(i));
		Status_Log:=2;

		TCount:=0;
		Timer(IN:=FALSE);
	END_IF
END_IF
(* Check timer *)
IF Timer.Q THEN
	TCount:=0;							(* One hour is elapsed *)
	IF TCount<Plant_MaxWaterLoss THEN
		Status_Log:=0;
	END_IF
END_IF
END_FUNCTION_BLOCK

(* POU Plant_Objects/obj_MBUS, ST *)
FUNCTION_BLOCK obj_MBUS
(* === M-BUS PROTOCOL INTERFACE ===
   v1.0[16/03/15] - Added interface errors
*)
VAR_INPUT
	(* Settings *)
	ID				: BYTE;
	COM				: BYTE;
	BAUDRATE		: COM_BAUDRATE;
	(* Interface *)
	MBus 			: typMBus;
	MBus_Master 	: FbMBusMaster;
END_VAR
VAR_OUTPUT
	(* Status *)
	Status_Log		: BYTE;
	Status_Vis 		: DWORD;
END_VAR
VAR
	Alarm			: FLT_EVENT;
END_VAR
MBus_Master( bCOMPORT:=COM , enumBAUDRATE:=BAUDRATE , utMBus:=MBus );

(* Check status *)
Alarm(IN:=(MBus.bCOM_ERROR<>0));
IF Alarm.EVH THEN
	LogEv(EL_Alarm,EO_MBUS,ID,1,BYTE_TO_STRING(MBus.bCOM_ERROR));
END_IF
IF Alarm.EVL THEN
	LogEv(EL_Log,EO_MBUS,ID,2,'MBUS_OK');
END_IF

(* Log/visu status *)
   IF Alarm.IN   					THEN Status_Log:=2; Status_Vis:=COLOR_RED;
ELSIF (MBus.bL1_ERROR AND 16#1F)<>0 THEN Status_Log:=1; Status_Vis:=COLOR_YELLOW;
  				 					ELSE Status_Log:=0; Status_Vis:=COLOR_GREEN;
END_IF
END_FUNCTION_BLOCK

(* POU Plant_Objects/obj_MBUS_CTB_SHARKY775, ST *)
FUNCTION_BLOCK obj_MBUS_CTB_SHARKY775
(* === M-BUS CONTABILIZER SHARKY 775 ===
   v1.0[16/03/15] - Error management
*)
VAR_INPUT
	(* Settings *)
	ID				: BYTE;
	ADDRESS			: DWORD;
	Refresh_Period	: TIME:=t#3m;
	(* Controls *)
	Refresh_Auto	: BOOL:=TRUE; (* Enable automatic refresh *)
	Refresh_Now		: BOOL; 	  (* Force an immediate refresh *)
END_VAR
VAR_IN_OUT
	(* Interface *)
	MBUS			: obj_MBUS;
END_VAR
VAR_OUTPUT
	M1				: FbMBus_Heat;
	(* Status *)
	Status_Log		: BYTE;
	Status_Vis 	 	: DWORD;
END_VAR
VAR
	dly 	 	: TON := (PT:=t#5s);
	M1_Start	: BOOL;

	init_st		: BOOL;
	bus_st0		: BYTE;
	dev_st0		: BYTE;

(*	S1			: FbMBusSend;
	S1_Start	: BOOL;*)
(*	C1			: FbUnitConverter; *)

END_VAR
(* Auto refresh timer *)
dly(IN:=NOT (dly.Q OR Refresh_Now OR (NOT Refresh_Auto)));
(* Trigger refresh *)
IF dly.Q OR Refresh_Now THEN
	dly.PT:=Refresh_Period;
	Refresh_Now:=FALSE;
	(* Start reading *)
	M1.dwAdr:= ADDRESS;
	M1.xSND_NKE:=TRUE;
	M1_Start:=TRUE;
END_IF

(* Contabilizer module *)
M1(	utMBus:=MBUS.MBus, xStart:=M1_Start );

(* Extra actions *)
(*C1( utMBus:=MBUS.MBus, xStart:=C1_Start );*)

(* Check status *)
IF NOT init_st OR M1.bError<>bus_st0 OR M1.utMBInfo.bMStatus<>dev_st0 THEN
	init_st:=TRUE;
	bus_st0:=M1.bError; dev_st0:=M1.utMBInfo.bMStatus;
	IF bus_st0<>0 THEN
		LogEv(EL_Alarm,EO_CTB,ID,2,BYTE_TO_STRING(bus_st0));
		Status_Log:=2; Status_Vis:=COLOR_RED;
	ELSE
		IF dev_st0<>0 THEN
			Status_Log:=2; Status_Vis:=COLOR_RED;
			CASE dev_st0 OF
				16#08: LogEv(EL_Alarm,EO_CTB,ID,10,'C-1');
				16#04: LogEv(EL_Alarm,EO_CTB,ID,10,'E-8');
				16#28: LogEv(EL_Alarm,EO_CTB,ID,10,'E-4');
				16#50: LogEv(EL_Alarm,EO_CTB,ID,10,'E-1');
				16#70: LogEv(EL_Alarm,EO_CTB,ID,10,'E-7');
				16#84: LogEv(EL_Alarm,EO_CTB,ID,10,'E-9');
				16#B0: LogEv(EL_Wrn  ,EO_CTB,ID,10,'E-3');
				16#D0: LogEv(EL_Wrn  ,EO_CTB,ID,10,'E-6');
				16#F0: LogEv(EL_Alarm,EO_CTB,ID,10,'Leak');
				16#10: LogEv(EL_Wrn  ,EO_CTB,ID,10,'E-5'); Status_Log:=1; Status_Vis:=COLOR_YELLOW;
			ELSE
				LogEv(EL_Alarm,EO_CTB,ID,10,BYTE_TO_STRING(dev_st0));
			END_CASE
		ELSE
			Status_Log:=0; Status_Vis:=16#20F020;
			LogEv(EL_Log,EO_CTB,ID,1,'');
		END_IF
	END_IF
END_IF

Lamp.obj_Status := Status_Log;
Lamp.UpdateStatus();
END_FUNCTION_BLOCK
ACTION AddLogData:
Logger.s1:=INSERT('&CTB=',BYTE_TO_STRING(ID),4);
IF ID<10 THEN Logger.s1:=INSERT(Logger.s1,'0',4); END_IF

Logger.s1:=CONCAT(Logger.s1,M1.utFTemp.Value);		Logger.s1:=CONCAT(Logger.s1,';');
Logger.s1:=CONCAT(Logger.s1,M1.utRTemp.Value);		Logger.s1:=CONCAT(Logger.s1,';');
Logger.s1:=CONCAT(Logger.s1,M1.utFlow.Value);		Logger.s1:=CONCAT(Logger.s1,';');
Logger.s1:=CONCAT(Logger.s1,M1.utPower.Value);		Logger.s1:=CONCAT(Logger.s1,';');
Logger.s1:=CONCAT(Logger.s1,M1.utEnergy.Value);		Logger.s1:=CONCAT(Logger.s1,';');

Logger.s1:=CONCAT(Logger.s1,BYTE_TO_STRING(Status_Log));
ADDSTRING(ADR(Logger.TData), ADR(Logger.s1), Logger.TLen);
END_ACTION

(* POU Plant_Objects/obj_MODBUS, ST *)
FUNCTION_BLOCK obj_MODBUS
(* === MODBUS PROTOCOL INTERFACE ===
   v1.1[19/06/15] - Added new VARS allocation and searching
*)
VAR CONSTANT
	VARS_Max	: BYTE := 32;
END_VAR
VAR_INPUT
	(* Settings *)
	ID			: BYTE;
	COM			: BYTE;
	BAUDRATE	: COM_BAUDRATE;
	RS485		: BOOL := FALSE;

	(* Interface *)
	MB_MASTER	: MODBUS_EXTENDED_MASTER;
	MB_Start	: BOOL;
	MB_Query	: typModbusExtendedQuery;
	MB_Resp		: typModbusResponse;
	MB_Lock		: BOOL;

	(* Variables management *)
	VARS_En		: BOOL;
	VARS		: ARRAY [0..VARS_Max] OF typ_MODBUS_VAR;
	VARS_Check	: BOOL;
	VARS_Alarm	: BOOL;

	(* Variables allocation *)
	VAR_Pointer : POINTER TO ARRAY[0..99] OF WORD;
	VAR_Cfg		: POINTER TO typ_MODBUS_VAR;
END_VAR
VAR_OUTPUT
	(* Status *)
	Status_Log	: BYTE;
	Status_Vis	: DWORD;
END_VAR
VAR
	sta         : BYTE :=0;
	i			: BYTE;
	j			: BYTE;
	Alarm		: FLT_EVENT;
	
	VarTmr		: TON := (PT:=T#1s);
	VarSta		: BYTE; (* Status *)
	VarCnt		: BYTE; (* Scan counter *)
	VarRetry	: BYTE;
	VarAlarm	: BYTE; (* Last variable with errors *)
END_VAR
MB_MASTER(ENABLE:=TRUE,	ASCII_Mode:=FALSE, bCOM_PORT:=COM, cbCOM_BAUDRATE:=BAUDRATE, cpCOM_PARITY:=PARITY_NO,
		csCOM_STOPBITS:=STOPBITS_1,	cbsCOM_BYTESIZE:=BS_8, cfCOM_FLOW_CONTROL:=SEL(RS485,NO_FLOW_CONTROL,HALFDUPLEX),
		tTIME_OUT:=t#250ms,	StartFunction:=MB_Start, ExtQuery:=MB_Query, Response:=MB_Resp);

(* Process variable management *)
IF VARS_En THEN VARS_Process(); END_IF

(* Check status *)
Alarm(IN:=(MB_MASTER.bInterfaceError<>0));
IF Alarm.EVH THEN
	LogEv(SEL(MB_MASTER.bInterfaceError<>3,EL_Wrn,EL_Alarm),EO_MODBUS,ID,1,BYTE_TO_STRING(MB_MASTER.bInterfaceError));
END_IF
IF Alarm.EVL THEN								(* Trigger a fall edge: MODBUS back working *)
	LogEv(EL_Log,EO_MODBUS,ID,2,'MODBUS_OK');
END_IF

(* Log/visu status *)
   IF Alarm.IN   THEN Status_Log:=2; Status_Vis:=COLOR_RED;
ELSIF Vars_Alarm THEN Status_Log:=1; Status_Vis:=COLOR_YELLOW;
  				 ELSE Status_Log:=0; Status_Vis:=COLOR_GREEN;
END_IF
END_FUNCTION_BLOCK
ACTION VAR_Search:
(* Search VAR with specific pointer if not found return first free VAR
	[Last VAR is not active... used as safe area...] 
*)
j:=VARS_Max;
FOR i := 0 TO VARS_Max-1 DO
	IF VARS[i].Variable=0 AND j>i THEN j:=i; END_IF
	IF VARS[i].Variable=VAR_Pointer THEN
		VAR_Cfg:=ADR(VARS[i]);
		RETURN;
	END_IF
END_FOR
VAR_Cfg:=ADR(VARS[j]);
END_ACTION
ACTION VARS_Process:
(* Update var timers *)
VarTmr(IN:=(NOT VarTmr.Q));
IF VarTmr.Q THEN
	FOR i := 0 TO VARS_Max DO
		IF VARS[i].Refresh_Cnt>0 THEN VARS[i].Refresh_Cnt:=VARS[i].Refresh_Cnt-1; END_IF
	END_FOR
	VARS_Check:=TRUE;
END_IF


(* Process status *)
CASE VarSta OF
	0: (* === Init *)
		VarCnt:=0;
		VarSta:=1;

	1: (* === Wait check signal *)
		IF VARS_Check THEN				(* Decremented "Refresh_Cnt" *)
			VARS_Check:=FALSE;
			VarCnt:=0;
			VarSta:=2;
		END_IF

	2: (* === Check loop *)
		IF NOT (MB_Lock OR MB_Start) THEN
			WHILE VarCnt<=(VARS_Max-1) AND VarSta=2 DO
				(* Check only active vars *)
				IF VARS[VarCnt].Variable<>0 THEN			(* "Variable" is a pointer to word, so if 0 no address *)
					(* Check var auto-refresh on timer checks *)
					IF VARS[VarCnt].Refresh_Time>0 AND VARS[VarCnt].Refresh_Cnt=0 THEN
						VARS[VarCnt].Refresh_Cnt:=VARS[VarCnt].Refresh_Time;
						VarSta:=3;
					END_IF
					(* Check refresh for change or request *)
					CASE VARS[VarCnt].FunCode OF
						5,6,15,16: (* Write functions *)
							IF VARS[VarCnt].Variable_Size=1 THEN
								IF VARS[VarCnt].Variable^<>VARS[VarCnt].Variable_Mirror THEN
									VARS[VarCnt].Variable_Mirror:=VARS[VarCnt].Variable^;
									VarSta:=3;
								END_IF
							ELSE
								IF VARS[VarCnt].Variable_Mirror<>0 THEN
									VARS[VarCnt].Variable_Mirror:=0;
									VarSta:=3;
								END_IF
							END_IF
						1,2,3,4: (* Read functions *)
							IF VARS[VarCnt].Variable_Mirror<>0 THEN
								VARS[VarCnt].Variable_Mirror:=0;
								VarSta:=3;
							END_IF
					END_CASE
				END_IF
				(* Process query *)
				IF VarSta=3 THEN
					MB_Lock:=TRUE;
					MB_Query.SlaveAddress:=VARS[VarCnt].SlaveAddress;
					MB_Query.FunctionCode:=VARS[VarCnt].FunCode;
					CASE VARS[VarCnt].FunCode OF
						16#5,16#6,16#F,16#10:
							MB_Query.Read_Quantity:=0;
							MB_Query.Read_StartAddress:=0;
							MB_Query.Write_StartAddress:=VARS[VarCnt].FunAddress;
							MB_Query.Write_Quantity:=VARS[VarCnt].Variable_Size;
							IF VARS[VarCnt].Variable_Size=200 THEN
								COPY_32SWAP16(VARS[VarCnt].Variable, ADR(MB_Query.Write_Data[0]));
							ELSIF VARS[VarCnt].Variable_Size>1 THEN
								MEMCPY(VARS[VarCnt].Variable, ADR(MB_Query.Write_Data[0]), 2*VARS[VarCnt].Variable_Size);
							ELSE
								MB_Query.Write_Data[0]:=VARS[VarCnt].Variable^;
							END_IF
						16#1,16#2,16#3,16#4:
							MB_Query.Read_StartAddress:=VARS[VarCnt].FunAddress;
							IF VARS[VarCnt].Variable_Size=200 THEN MB_Query.Read_Quantity:=2; ELSE
							  MB_Query.Read_Quantity:=VARS[VarCnt].Variable_Size;
							END_IF
							MB_Query.Write_StartAddress:=0;
							MB_Query.Write_Quantity:=0;
					END_CASE
					VarRetry:=0;
					MB_Start:=TRUE;
				ELSE
					VarCnt:=VarCnt+1;
				END_IF
			END_WHILE
			(* Check loop completed -> no actions *)
			IF VarSta=2 THEN VarSta:=1; END_IF
		END_IF

	3: (* === Wait & process MB response *)
		IF NOT MB_Start THEN
			IF MB_MASTER.MB_Error=0 THEN
				CASE VARS[VarCnt].FunCode OF
					1,2,3,4:
						IF VARS[VarCnt].Variable_Size=200 THEN
							COPY_32SWAP16(ADR(MB_Resp.Data), VARS[VarCnt].Variable);
						ELSIF VARS[VarCnt].Variable_Size>1 THEN
							MEMCPY(ADR(MB_Resp.Data), VARS[VarCnt].Variable, 2*VARS[VarCnt].Variable_Size);
						ELSE
							VARS[VarCnt].Variable^:=MB_Resp.Data[0];
						END_IF
				END_CASE
				MB_Lock:=FALSE;
				(* Signal error recovery *)
				IF VARS_Alarm=TRUE AND VarCnt=VarAlarm THEN
					LogEv(EL_Wrn,EO_MODBUS,ID,5,'');
					VARS_Alarm:=FALSE;
				END_IF
				(* Next var *)
				VarCnt:=VarCnt+1;
				VarSta:=2;
			ELSE
				IF VarRetry<3 THEN
					VarRetry:=VarRetry+1;
					MB_Start:=TRUE;
				ELSE
					MB_Lock:=FALSE;
					(* Signal error *)
					IF VARS_Alarm=FALSE THEN
						LogEv(EL_Wrn,EO_MODBUS,ID,3,INT_TO_STRING(MB_MASTER.MB_Error));
						VARS_Alarm:=TRUE;
						VarAlarm:=VarCnt-1;
					END_IF
					(* Next var *)
					VarCnt:=VarCnt+1;
					VarSta:=2;
				END_IF
			END_IF
		END_IF

ELSE
	VarSta:=0;
END_CASE
END_ACTION

(* POU Plant_Objects/obj_MODBUS_CIR, ST *)
FUNCTION_BLOCK obj_MODBUS_CIR
VAR CONSTANT
	WAIT_STATE		:	BYTE := 0;
	PUMP_STATUS		:	BYTE := 1;
	PUMP_DATA		:	BYTE := 2;
	PUMP_ALARMS		:	BYTE := 3;
	PUMP_END_READ	:	BYTE := 4;
	CIR_ON_OFF		:	BYTE := 90;
	CIR_ON_OFF_CHECK:	BYTE := 91;
	CIR_END_WRITE	:	BYTE := 92;
	ERROR_STATE		:	BYTE := 100;
END_VAR
VAR_INPUT
	ID		:	BYTE;
	Address :	BYTE;		(* Pump address *)

	(* Controls *)
	Ctrl_SetPoint 	: INT;
	CIR_RUN_REQ		: BOOL; (* External run request (no heat or cold requested) *)
	CIR_STOP_REQ	: BOOL; (* External stop request (has priority over RUN signals!) *)

	CIR_AL			: BOOL; (* Alarm input signal *)
	CIR_AUTO		: BOOL;

	OnOff			: BYTE;
END_VAR
VAR_IN_OUT
	ModBus		:	obj_MODBUS;
END_VAR
VAR_OUTPUT
	Run			:	BOOL;

	Status_Log	:	WORD;
	Status_Vis	:	DWORD;
END_VAR
VAR
	Ctrl_Run	:	BOOL;		(* Logical status of the device: 0: Not running (switched off), 1: running *)
	CirStatus	:	BYTE;
	OldCirStatus:	BYTE;
	fWrite		:	BOOL;

	state		:	BYTE;
	retry		:	BYTE;
	ReadTmr		:	TON := (PT:=T#5m);
	retry_write	:	BYTE;

	DataPump	:	typ_MODBUS_CIR;

	OldAlarm	:	WORD;

	fWrn		:	BOOL;

	fStatus		:	FLT_EVENT;
	fCIR_AUTO	:	FLT_EVENT;
	Alarm		:	FLT_EVENT;
	AlarmHw		:	FLT_EVENT := (INITEV:=FALSE);
	Inverter	:	FLT_EVENT := (INITEV:=FALSE);
	Warning		:	FLT_EVENT := (INITEV:=FALSE);

	s1			:	STRING;
	Delay		: 	TONOF := (PT_OF:=Plant_CirOffDelay);
END_VAR
ManagePump();

(* State machine to read pump parameters *)
Stm();

(* Check alarm and warning for both pumps *)
CheckFault();

IF Status_Log = 2 THEN Run := FALSE;
ELSE Run := Ctrl_Run;
END_IF

Lamp.obj_Status := Status_Log;
Lamp.UpdateStatus();

IF Status_Log = 2 THEN Status_Vis := COLOR_RED;
ELSIF Status_Log = 1 THEN Status_Vis := COLOR_YELLOW;
ELSE Status_Vis := COLOR_GREEN;
END_IF
END_FUNCTION_BLOCK
ACTION AddLogData:
Logger.s1:=INSERT('&CIR=',BYTE_TO_STRING(ID),4);
IF ID<10 THEN Logger.s1:=INSERT(Logger.s1,'0',4); END_IF

Logger.s1:=CONCAT(Logger.s1,WORD_TO_STRING(DataPump.PumpStatus));		Logger.s1:=CONCAT(Logger.s1,';');
Logger.s1:=CONCAT(Logger.s1,INT_TO_STRING(DataPump.PumpBoardTemp));		Logger.s1:=CONCAT(Logger.s1,';');
Logger.s1:=CONCAT(Logger.s1,WORD_TO_STRING(DataPump.PumpVoltage));		Logger.s1:=CONCAT(Logger.s1,';');
Logger.s1:=CONCAT(Logger.s1,WORD_TO_STRING(DataPump.PumpRPM));			Logger.s1:=CONCAT(Logger.s1,';');
Logger.s1:=CONCAT(Logger.s1,WORD_TO_STRING(DataPump.PumpPower));		Logger.s1:=CONCAT(Logger.s1,';');
Logger.s1:=CONCAT(Logger.s1,DWORD_TO_STRING(DataPump.PumpOpTime));		Logger.s1:=CONCAT(Logger.s1,';');
Logger.s1:=CONCAT(Logger.s1,WORD_TO_STRING(DataPump.PumpHead));			Logger.s1:=CONCAT(Logger.s1,';');
Logger.s1:=CONCAT(Logger.s1,WORD_TO_STRING(DataPump.PumpFlow));			Logger.s1:=CONCAT(Logger.s1,';');
Logger.s1:=CONCAT(Logger.s1,WORD_TO_STRING(DataPump.PumpLiqTemp));		Logger.s1:=CONCAT(Logger.s1,';');

Logger.s1:=CONCAT(Logger.s1,WORD_TO_STRING(Status_Log));
ADDSTRING(ADR(Logger.TData), ADR(Logger.s1), Logger.TLen);
END_ACTION
ACTION CheckFault:
AlarmHw(IN:=CIR_AL);

IF AlarmHw.EVH THEN
	LogEv(EL_Alarm,EO_CIR,ID,3,'CIR_Alarm');
	Status_Log := 2;
END_IF

IF AlarmHw.EVL THEN
	LogEv(EL_Alarm,EO_CIR,ID,4,'CIR_Alarm_Recovered');
	Status_Log := 0;
END_IF

Inverter(IN:=DataPump.PumpFault);

IF Inverter.EVH THEN
	LogEv(EL_Alarm,EO_CIR,ID,9,'Inverter_Fault');
	Status_Log := 2;
END_IF

IF Inverter.EVL THEN
	LogEv(EL_Alarm,EO_CIR,ID,10,'Inverter_Fault_Recovered');
	Status_Log := 0;
END_IF

Alarm(IN:=(DataPump.PumpAlarm[0] <> OldAlarm));

IF Alarm.EVH THEN
	IF DataPump.PumpAlarm[0] = 0 THEN
		LogEv(EL_Alarm,EO_CIR,ID,12,'Alarm_Recovered');
		Status_Log := 0;
	ELSE
		s1 := WORD_TO_STRING(DataPump.PumpAlarm[0]);
		LogEv(EL_Alarm,EO_CIR,ID,11,s1);
		Status_Log := 2;
	END_IF

	OldAlarm := DataPump.PumpAlarm[0];
END_IF

IF DataPump.PumpLiqTemp < 5 OR DataPump.PumpLiqTemp > 80 THEN fWrn := TRUE;
ELSE fWrn := FALSE;
END_IF

Warning(IN:=fWrn);

IF Warning.EVH THEN
	LogEv(EL_Wrn,EO_CIR,ID,13,'Liquid_Temperature');

	IF Status_Log <> 2 THEN Status_Log := 1; END_IF
END_IF

IF Warning.EVL THEN
	LogEv(EL_Log,EO_CIR,ID,14,'Liquid_Temperature_Recovered');
	Status_Log := 0;
END_IF
END_ACTION
ACTION ManagePump:
(* Copy actual status as old status *)
OldCirStatus := CirStatus;

fCIR_AUTO(IN:=CIR_AUTO);
IF fCIR_AUTO.EVL THEN
	LogEv(EL_Wrn,EO_CIR,ID,7,'CIR_Manual');

	(* MANUAL MODE	-> CIR working depends on external signal *)
	CirStatus := 2;
	fWrite := TRUE;

END_IF

IF fCIR_AUTO.EVH THEN LogEv(EL_Log,EO_CIR,ID,8,'CIR_Auto'  ); END_IF

(* AUTOMATIC MODE *)
IF CIR_AUTO THEN

	IF OnOff = 0 THEN
	
		Ctrl_Run := FALSE;			(* Logically swtched off *)
		Delay(IN:=Ctrl_Run);		(* Count delay time before physical switch off	*)

	ELSIF OnOff = 1 THEN

		(* Start switch on delay time (proportional to object id) *)
		Delay(IN:=TRUE, PT_ON:=WORD_TO_TIME(1000*ID));
	
